LIN {X 0,Y 641.804,Z 360.991,A -85,B 0,C 180,E1 23081.821,E2 23081.821} C_VEL
LIN {X 0,Y 635.223,Z 347.429,A -85,B 0,C 180,E1 23079.954,E2 23079.954} C_VEL
LIN {X 0,Y 631.078,Z 339.172,A -85,B 0,C 180,E1 23078.744,E2 23078.744} C_VEL
LIN {X 0,Y 626.769,Z 330.556,A -85,B 0,C 180,E1 23077.432,E2 23077.432} C_VEL
LIN {X 0,Y 625.015,Z 327.05,A -85,B 0,C 180,E1 23076.864,E2 23076.864} C_VEL
LIN {X 0,Y 624.908,Z 326.441,A -85,B 0,C 180,E1 23076.643,E2 23076.643} C_VEL
LIN {X 0,Y 624.949,Z 326.345,A -85,B 0,C 180,E1 23073.503,E2 23073.503} C_VEL
LIN {X 0,Y 624.913,Z 326.377,A -85,B 0,C 180,E1 23070.412,E2 23070.412} C_VEL
LIN {X 0,Y 624.947,Z 326.372,A -85,B 0,C 180,E1 23067.232,E2 23067.232} C_VEL
LIN {X 0,Y 624.931,Z 326.347,A -85,B 0,C 180,E1 23064.079,E2 23064.079} C_VEL
LIN {X 0,Y 624.933,Z 326.384,A -85,B 0,C 180,E1 23060.806,E2 23060.806} C_VEL
LIN {X 0,Y 624.947,Z 326.347,A -85,B 0,C 180,E1 23057.698,E2 23057.698} C_VEL
LIN {X 0,Y 624.931,Z 326.381,A -85,B 0,C 180,E1 23054.537,E2 23054.537} C_VEL
LIN {X 0,Y 624.939,Z 326.352,A -85,B 0,C 180,E1 23051.443,E2 23051.443} C_VEL
LIN {X 0,Y 624.935,Z 326.375,A -85,B 0,C 180,E1 23048.372,E2 23048.372} C_VEL
LIN {X 0,Y 624.93,Z 326.352,A -85,B 0,C 180,E1 23045.325,E2 23045.325} C_VEL
LIN {X 0,Y 624.94,Z 326.376,A -85,B 0,C 180,E1 23042.201,E2 23042.201} C_VEL
LIN {X 0,Y 624.923,Z 326.355,A -85,B 0,C 180,E1 23039.083,E2 23039.083} C_VEL
LIN {X 0,Y 624.944,Z 326.376,A -85,B 0,C 180,E1 23035.963,E2 23035.963} C_VEL
LIN {X 0,Y 624.915,Z 326.354,A -85,B 0,C 180,E1 23032.923,E2 23032.923} C_VEL
LIN {X 0,Y 624.949,Z 326.375,A -85,B 0,C 180,E1 23029.863,E2 23029.863} C_VEL
LIN {X 0,Y 624.908,Z 326.359,A -85,B 0,C 180,E1 23026.773,E2 23026.773} C_VEL
LIN {X 0,Y 624.953,Z 326.368,A -85,B 0,C 180,E1 23023.73,E2 23023.73} C_VEL
LIN {X 0,Y 624.903,Z 326.37,A -85,B 0,C 180,E1 23020.657,E2 23020.657} C_VEL
LIN {X 0,Y 624.955,Z 326.352,A -85,B 0,C 180,E1 23017.618,E2 23017.618} C_VEL
LIN {X 0,Y 624.896,Z 326.392,A -85,B 0,C 180,E1 23014.607,E2 23014.607} C_VEL
LIN {X 0,Y 624.957,Z 326.344,A -85,B 0,C 180,E1 23011.629,E2 23011.629} C_VEL
LIN {X 0,Y 624.888,Z 326.373,A -85,B 0,C 180,E1 23008.665,E2 23008.665} C_VEL
LIN {X 0,Y 624.913,Z 326.378,A -85,B 0,C 180,E1 23005.813,E2 23005.813} C_VEL
LIN {X 0,Y 624.927,Z 326.63,A -85,B 0,C 180,E1 23004.753,E2 23004.753} C_VEL
LIN {X 0,Y 626.262,Z 329.964,A -85,B 0,C 180,E1 23004.242,E2 23004.242} C_VEL
LIN {X 0,Y 627.651,Z 332.24,A -85,B 0,C 180,E1 23003.869,E2 23003.869} C_VEL
LIN {X 0,Y 630.344,Z 337.573,A -85,B 0,C 180,E1 23003.079,E2 23003.079} C_VEL
LIN {X 0,Y 636.416,Z 349.11,A -85,B 0,C 180,E1 23001.41,E2 23001.41} C_VEL
LIN {X 0,Y 638.709,Z 353.459,A -85,B 0,C 180,E1 23000.855,E2 23000.855} C_VEL
LIN {X 0,Y 656.316,Z 378.29,A -85,B 0,C 180,E1 22998.74,E2 22998.74} C_VEL
LIN {X 0,Y 661.405,Z 385.767,A -85,B 0,C 180,E1 22998.161,E2 22998.161} C_VEL
LIN {X 0,Y 657.846,Z 584.34,A -85,B 0,C 180,E1 22995.477,E2 22995.477} C_VEL
LIN {X 0,Y 653.631,Z 808.573,A -85,B 0,C 180,E1 22992.489,E2 22992.489} C_VEL
LIN {X 0,Y 652.607,Z 840.702,A -85,B 0,C 180,E1 22992.004,E2 22992.004} C_VEL
LIN {X 0,Y 651.456,Z 864.088,A -85,B 0,C 180,E1 22991.512,E2 22991.512} C_VEL
LIN {X 0,Y 650.123,Z 886.354,A -85,B 0,C 180,E1 22990.922,E2 22990.922} C_VEL
LIN {X 0,Y 648.327,Z 912.621,A -85,B 0,C 180,E1 22990.066,E2 22990.066} C_VEL
LIN {X 0,Y 646.181,Z 938.349,A -85,B 0,C 180,E1 22989.032,E2 22989.032} C_VEL
LIN {X 0,Y 644.374,Z 958.689,A -85,B 0,C 180,E1 22988.083,E2 22988.083} C_VEL
LIN {X 0,Y 642.408,Z 979.352,A -85,B 0,C 180,E1 22986.988,E2 22986.988} C_VEL
LIN {X 0,Y 639.991,Z 1003.732,A -85,B 0,C 180,E1 22985.512,E2 22985.512} C_VEL
LIN {X 0,Y 637.696,Z 1025.632,A -85,B 0,C 180,E1 22983.979,E2 22983.979} C_VEL
LIN {X 0,Y 635.819,Z 1043.504,A -85,B 0,C 180,E1 22982.583,E2 22982.583} C_VEL
LIN {X 0,Y 633.971,Z 1061.27,A -85,B 0,C 180,E1 22981.046,E2 22981.046} C_VEL
LIN {X 0,Y 631.756,Z 1082.664,A -85,B 0,C 180,E1 22978.967,E2 22978.967} C_VEL
LIN {X 0,Y 630.187,Z 1098.843,A -85,B 0,C 180,E1 22977.19,E2 22977.19} C_VEL
LIN {X 0,Y 628.766,Z 1114.163,A -85,B 0,C 180,E1 22975.326,E2 22975.326} C_VEL
LIN {X 0,Y 627.338,Z 1131.25,A -85,B 0,C 180,E1 22972.985,E2 22972.985} C_VEL
LIN {X 0,Y 626.314,Z 1144.859,A -85,B 0,C 180,E1 22970.855,E2 22970.855} C_VEL
LIN {X 0,Y 625.553,Z 1156.307,A -85,B 0,C 180,E1 22968.837,E2 22968.837} C_VEL
LIN {X 0,Y 624.897,Z 1168.201,A -85,B 0,C 180,E1 22966.452,E2 22966.452} C_VEL
LIN {X 0,Y 624.452,Z 1178.088,A -85,B 0,C 180,E1 22964.086,E2 22964.086} C_VEL
LIN {X 0,Y 624.187,Z 1185.798,A -85,B 0,C 180,E1 22961.926,E2 22961.926} C_VEL
LIN {X 0,Y 624.035,Z 1192.621,A -85,B 0,C 180,E1 22959.592,E2 22959.592} C_VEL
LIN {X 0,Y 623.952,Z 1198.251,A -85,B 0,C 180,E1 22957.088,E2 22957.088} C_VEL
LIN {X 0,Y 623.914,Z 1202.013,A -85,B 0,C 180,E1 22954.688,E2 22954.688} C_VEL
LIN {X 0,Y 623.909,Z 1204.208,A -85,B 0,C 180,E1 22952.388,E2 22952.388} C_VEL
LIN {X 0,Y 623.902,Z 1204.961,A -85,B 0,C 180,E1 22949.816,E2 22949.816} C_VEL
LIN {X 0,Y 623.908,Z 1204.072,A -85,B 0,C 180,E1 22947.428,E2 22947.428} C_VEL
LIN {X 0,Y 623.916,Z 1201.898,A -85,B 0,C 180,E1 22945.22,E2 22945.22} C_VEL
LIN {X 0,Y 623.957,Z 1198.078,A -85,B 0,C 180,E1 22942.819,E2 22942.819} C_VEL
LIN {X 0,Y 624.037,Z 1192.376,A -85,B 0,C 180,E1 22940.314,E2 22940.314} C_VEL
LIN {X 0,Y 624.193,Z 1185.493,A -85,B 0,C 180,E1 22937.98,E2 22937.98} C_VEL
LIN {X 0,Y 624.484,Z 1177.37,A -85,B 0,C 180,E1 22935.725,E2 22935.725} C_VEL
LIN {X 0,Y 624.975,Z 1166.372,A -85,B 0,C 180,E1 22933.167,E2 22933.167} C_VEL
LIN {X 0,Y 625.583,Z 1155.793,A -85,B 0,C 180,E1 22931.067,E2 22931.067} C_VEL
LIN {X 0,Y 626.354,Z 1144.276,A -85,B 0,C 180,E1 22929.048,E2 22929.048} C_VEL
LIN {X 0,Y 627.501,Z 1129.294,A -85,B 0,C 180,E1 22926.723,E2 22926.723} C_VEL
LIN {X 0,Y 628.841,Z 1113.387,A -85,B 0,C 180,E1 22924.576,E2 22924.576} C_VEL
LIN {X 0,Y 630.262,Z 1097.992,A -85,B 0,C 180,E1 22922.711,E2 22922.711} C_VEL
LIN {X 0,Y 632.179,Z 1078.816,A -85,B 0,C 180,E1 22920.633,E2 22920.633} C_VEL
LIN {X 0,Y 634.138,Z 1059.603,A -85,B 0,C 180,E1 22918.804,E2 22918.804} C_VEL
LIN {X 0,Y 635.95,Z 1042.219,A -85,B 0,C 180,E1 22917.311,E2 22917.311} C_VEL
LIN {X 0,Y 637.972,Z 1022.949,A -85,B 0,C 180,E1 22915.82,E2 22915.82} C_VEL
LIN {X 0,Y 640.482,Z 998.662,A -85,B 0,C 180,E1 22914.167,E2 22914.167} C_VEL
LIN {X 0,Y 642.581,Z 977.633,A -85,B 0,C 180,E1 22912.917,E2 22912.917} C_VEL
LIN {X 0,Y 644.476,Z 957.681,A -85,B 0,C 180,E1 22911.867,E2 22911.867} C_VEL
LIN {X 0,Y 646.516,Z 934.93,A -85,B 0,C 180,E1 22910.819,E2 22910.819} C_VEL
LIN {X 0,Y 648.637,Z 907.797,A -85,B 0,C 180,E1 22909.767,E2 22909.767} C_VEL
LIN {X 0,Y 650.225,Z 884.749,A -85,B 0,C 180,E1 22909.032,E2 22909.032} C_VEL
LIN {X 0,Y 651.542,Z 862.576,A -85,B 0,C 180,E1 22908.452,E2 22908.452} C_VEL
LIN {X 0,Y 652.811,Z 836.723,A -85,B 0,C 180,E1 22907.922,E2 22907.922} C_VEL
LIN {X 0,Y 653.818,Z 798.385,A -85,B 0,C 180,E1 22907.377,E2 22907.377} C_VEL
LIN {X 0,Y 658.111,Z 571.161,A -85,B 0,C 180,E1 22904.345,E2 22904.345} C_VEL
LIN {X 0,Y 661.359,Z 385.453,A -85,B 0,C 180,E1 22901.83,E2 22901.83} C_VEL
LIN {X 0,Y 644.698,Z 361.888,A -85,B 0,C 180,E1 22899.89,E2 22899.89} C_VEL
LIN {X 0,Y 638.077,Z 352.586,A -85,B 0,C 180,E1 22899.047,E2 22899.047} C_VEL
LIN {X 0,Y 633.374,Z 343.405,A -85,B 0,C 180,E1 22897.773,E2 22897.773} C_VEL
LIN {X 0,Y 628.853,Z 334.634,A -85,B 0,C 180,E1 22896.489,E2 22896.489} C_VEL
LIN {X 0,Y 626.609,Z 330.419,A -85,B 0,C 180,E1 22895.844,E2 22895.844} C_VEL
LIN {X 0,Y 624.978,Z 326.955,A -85,B 0,C 180,E1 22895.31,E2 22895.31} C_VEL
LIN {X 0,Y 624.918,Z 326.379,A -85,B 0,C 180,E1 22894.947,E2 22894.947} C_VEL
LIN {X 0,Y 624.888,Z 326.361,A -85,B 0,C 180,E1 22891.826,E2 22891.826} C_VEL
LIN {X 0,Y 624.899,Z 326.361,A -85,B 0,C 180,E1 22889.106,E2 22889.106} C_VEL
LIN {X 0,Y 624.906,Z 326.39,A -85,B 0,C 180,E1 22885.799,E2 22885.799} C_VEL
LIN {X 0,Y 624.915,Z 326.349,A -85,B 0,C 180,E1 22882.881,E2 22882.881} C_VEL
LIN {X 0,Y 624.911,Z 326.38,A -85,B 0,C 180,E1 22879.634,E2 22879.634} C_VEL
LIN {X 0,Y 624.94,Z 326.36,A -85,B 0,C 180,E1 22876.589,E2 22876.589} C_VEL
LIN {X 0,Y 624.912,Z 326.364,A -85,B 0,C 180,E1 22873.415,E2 22873.415} C_VEL
LIN {X 0,Y 624.949,Z 326.368,A -85,B 0,C 180,E1 22870.323,E2 22870.323} C_VEL
LIN {X 0,Y 624.914,Z 326.357,A -85,B 0,C 180,E1 22867.169,E2 22867.169} C_VEL
LIN {X 0,Y 624.947,Z 326.372,A -85,B 0,C 180,E1 22864.129,E2 22864.129} C_VEL
LIN {X 0,Y 624.919,Z 326.359,A -85,B 0,C 180,E1 22861.008,E2 22861.008} C_VEL
LIN {X 0,Y 624.941,Z 326.368,A -85,B 0,C 180,E1 22857.983,E2 22857.983} C_VEL
LIN {X 0,Y 624.927,Z 326.359,A -85,B 0,C 180,E1 22854.859,E2 22854.859} C_VEL
LIN {X 0,Y 624.935,Z 326.365,A -85,B 0,C 180,E1 22851.813,E2 22851.813} C_VEL
LIN {X 0,Y 624.934,Z 326.359,A -85,B 0,C 180,E1 22848.744,E2 22848.744} C_VEL
LIN {X 0,Y 624.93,Z 326.372,A -85,B 0,C 180,E1 22845.641,E2 22845.641} C_VEL
LIN {X 0,Y 624.939,Z 326.355,A -85,B 0,C 180,E1 22842.591,E2 22842.591} C_VEL
LIN {X 0,Y 624.926,Z 326.384,A -85,B 0,C 180,E1 22839.488,E2 22839.488} C_VEL
LIN {X 0,Y 624.944,Z 326.347,A -85,B 0,C 180,E1 22836.422,E2 22836.422} C_VEL
LIN {X 0,Y 624.92,Z 326.387,A -85,B 0,C 180,E1 22833.384,E2 22833.384} C_VEL
LIN {X 0,Y 624.947,Z 326.35,A -85,B 0,C 180,E1 22830.316,E2 22830.316} C_VEL
LIN {X 0,Y 624.908,Z 326.356,A -85,B 0,C 180,E1 22827.312,E2 22827.312} C_VEL
LIN {X 0,Y 624.954,Z 326.378,A -85,B 0,C 180,E1 22824.21,E2 22824.21} C_VEL
LIN {X 0,Y 624.946,Z 326.651,A -85,B 0,C 180,E1 22823.105,E2 22823.105} C_VEL
LIN {X 0,Y 626.468,Z 330.148,A -85,B 0,C 180,E1 22822.547,E2 22822.547} C_VEL
LIN {X 0,Y 627.637,Z 332.307,A -85,B 0,C 180,E1 22822.201,E2 22822.201} C_VEL
LIN {X 0,Y 634.063,Z 344.875,A -85,B 0,C 180,E1 22820.307,E2 22820.307} C_VEL
LIN {X 0,Y 641.872,Z 361.171,A -85,B 0,C 180,E1 22818.065,E2 22818.065} C_VEL
LIN {X 0,Y 649.819,Z 378.958,A -85,B 0,C 180,E1 22815.837,E2 22815.837} C_VEL
LIN {X 0,Y 648.792,Z 394.463,A -85,B 0,C 180,E1 22814.752,E2 22814.752} C_VEL
LIN {X 0,Y 650.304,Z 401.327,A -85,B 0,C 180,E1 22814.502,E2 22814.502} C_VEL
LIN {X 0,Y 651.352,Z 408.644,A -85,B 0,C 180,E1 22814.292,E2 22814.292} C_VEL
LIN {X 0,Y 651.333,Z 419.658,A -85,B 0,C 180,E1 22814.125,E2 22814.125} C_VEL
LIN {X 0,Y 650.372,Z 436.541,A -85,B 0,C 180,E1 22813.955,E2 22813.955} C_VEL
LIN {X 0,Y 645.669,Z 670.245,A -85,B 0,C 180,E1 22810.849,E2 22810.849} C_VEL
LIN {X 0,Y 642.293,Z 830.084,A -85,B 0,C 180,E1 22808.725,E2 22808.725} C_VEL
LIN {X 0,Y 641.163,Z 856.269,A -85,B 0,C 180,E1 22808.241,E2 22808.241} C_VEL
LIN {X 0,Y 639.753,Z 879.486,A -85,B 0,C 180,E1 22807.648,E2 22807.648} C_VEL
LIN {X 0,Y 638.346,Z 899.141,A -85,B 0,C 180,E1 22807.032,E2 22807.032} C_VEL
LIN {X 0,Y 636.661,Z 920.113,A -85,B 0,C 180,E1 22806.249,E2 22806.249} C_VEL
LIN {X 0,Y 634.578,Z 944.969,A -85,B 0,C 180,E1 22805.158,E2 22805.158} C_VEL
LIN {X 0,Y 632.686,Z 965.707,A -85,B 0,C 180,E1 22804.093,E2 22804.093} C_VEL
LIN {X 0,Y 630.876,Z 984.683,A -85,B 0,C 180,E1 22802.985,E2 22802.985} C_VEL
LIN {X 0,Y 628.583,Z 1007.653,A -85,B 0,C 180,E1 22801.45,E2 22801.45} C_VEL
LIN {X 0,Y 626.685,Z 1026.358,A -85,B 0,C 180,E1 22800.013,E2 22800.013} C_VEL
LIN {X 0,Y 624.97,Z 1043.343,A -85,B 0,C 180,E1 22798.556,E2 22798.556} C_VEL
LIN {X 0,Y 622.908,Z 1063.939,A -85,B 0,C 180,E1 22796.554,E2 22796.554} C_VEL
LIN {X 0,Y 621.441,Z 1079.527,A -85,B 0,C 180,E1 22794.831,E2 22794.831} C_VEL
LIN {X 0,Y 619.965,Z 1096.148,A -85,B 0,C 180,E1 22792.773,E2 22792.773} C_VEL
LIN {X 0,Y 618.758,Z 1110.872,A -85,B 0,C 180,E1 22790.667,E2 22790.667} C_VEL
LIN {X 0,Y 617.877,Z 1123.126,A -85,B 0,C 180,E1 22788.688,E2 22788.688} C_VEL
LIN {X 0,Y 617.093,Z 1136.012,A -85,B 0,C 180,E1 22786.279,E2 22786.279} C_VEL
LIN {X 0,Y 616.619,Z 1145.191,A -85,B 0,C 180,E1 22784.269,E2 22784.269} C_VEL
LIN {X 0,Y 616.299,Z 1153.404,A -85,B 0,C 180,E1 22782.176,E2 22782.176} C_VEL
LIN {X 0,Y 616.061,Z 1161.254,A -85,B 0,C 180,E1 22779.718,E2 22779.718} C_VEL
LIN {X 0,Y 615.977,Z 1166.228,A -85,B 0,C 180,E1 22777.743,E2 22777.743} C_VEL
LIN {X 0,Y 615.913,Z 1170.071,A -85,B 0,C 180,E1 22775.777,E2 22775.777} C_VEL
LIN {X 0,Y 615.902,Z 1173.027,A -85,B 0,C 180,E1 22773.63,E2 22773.63} C_VEL
LIN {X 0,Y 615.911,Z 1174.701,A -85,B 0,C 180,E1 22771.209,E2 22771.209} C_VEL
LIN {X 0,Y 615.901,Z 1174.814,A -85,B 0,C 180,E1 22769.163,E2 22769.163} C_VEL
LIN {X 0,Y 615.906,Z 1173.836,A -85,B 0,C 180,E1 22767.209,E2 22767.209} C_VEL
LIN {X 0,Y 615.921,Z 1171.322,A -85,B 0,C 180,E1 22764.878,E2 22764.878} C_VEL
LIN {X 0,Y 615.961,Z 1167.047,A -85,B 0,C 180,E1 22762.539,E2 22762.539} C_VEL
LIN {X 0,Y 616.053,Z 1162.263,A -85,B 0,C 180,E1 22760.565,E2 22760.565} C_VEL
LIN {X 0,Y 616.21,Z 1156.003,A -85,B 0,C 180,E1 22758.488,E2 22758.488} C_VEL
LIN {X 0,Y 616.555,Z 1146.792,A -85,B 0,C 180,E1 22756.017,E2 22756.017} C_VEL
LIN {X 0,Y 616.992,Z 1137.822,A -85,B 0,C 180,E1 22754.009,E2 22754.009} C_VEL
LIN {X 0,Y 617.591,Z 1127.457,A -85,B 0,C 180,E1 22751.988,E2 22751.988} C_VEL
LIN {X 0,Y 618.549,Z 1113.531,A -85,B 0,C 180,E1 22749.649,E2 22749.649} C_VEL
LIN {X 0,Y 619.608,Z 1100.314,A -85,B 0,C 180,E1 22747.715,E2 22747.715} C_VEL
LIN {X 0,Y 620.996,Z 1084.506,A -85,B 0,C 180,E1 22745.658,E2 22745.658} C_VEL
LIN {X 0,Y 622.612,Z 1067.07,A -85,B 0,C 180,E1 22743.69,E2 22743.69} C_VEL
LIN {X 0,Y 624.168,Z 1051.184,A -85,B 0,C 180,E1 22742.083,E2 22742.083} C_VEL
LIN {X 0,Y 626.351,Z 1029.845,A -85,B 0,C 180,E1 22740.181,E2 22740.181} C_VEL
LIN {X 0,Y 628.199,Z 1011.463,A -85,B 0,C 180,E1 22738.743,E2 22738.743} C_VEL
LIN {X 0,Y 630.281,Z 990.792,A -85,B 0,C 180,E1 22737.305,E2 22737.305} C_VEL
LIN {X 0,Y 632.479,Z 967.857,A -85,B 0,C 180,E1 22735.935,E2 22735.935} C_VEL
LIN {X 0,Y 634.238,Z 948.527,A -85,B 0,C 180,E1 22734.926,E2 22734.926} C_VEL
LIN {X 0,Y 636.336,Z 924.605,A -85,B 0,C 180,E1 22733.842,E2 22733.842} C_VEL
LIN {X 0,Y 638.238,Z 900.726,A -85,B 0,C 180,E1 22732.933,E2 22732.933} C_VEL
LIN {X 0,Y 639.672,Z 880.707,A -85,B 0,C 180,E1 22732.298,E2 22732.298} C_VEL
LIN {X 0,Y 640.897,Z 860.874,A -85,B 0,C 180,E1 22731.78,E2 22731.78} C_VEL
LIN {X 0,Y 642.142,Z 836.025,A -85,B 0,C 180,E1 22731.276,E2 22731.276} C_VEL
LIN {X 0,Y 643.231,Z 791.041,A -85,B 0,C 180,E1 22730.653,E2 22730.653} C_VEL
LIN {X 0,Y 647.657,Z 571.402,A -85,B 0,C 180,E1 22727.75,E2 22727.75} C_VEL
LIN {X 0,Y 650.402,Z 429.922,A -85,B 0,C 180,E1 22725.856,E2 22725.856} C_VEL
LIN {X 0,Y 642.675,Z 393.196,A -85,B 0,C 180,E1 22724.529,E2 22724.529} C_VEL
LIN {X 0,Y 643.362,Z 382.663,A -85,B 0,C 180,E1 22723.757,E2 22723.757} C_VEL
LIN {X 0,Y 635.717,Z 365.668,A -85,B 0,C 180,E1 22721.586,E2 22721.586} C_VEL
LIN {X 0,Y 629.219,Z 352.169,A -85,B 0,C 180,E1 22719.704,E2 22719.704} C_VEL
LIN {X 0,Y 625.087,Z 343.962,A -85,B 0,C 180,E1 22718.481,E2 22718.481} C_VEL
LIN {X 0,Y 621.118,Z 336.002,A -85,B 0,C 180,E1 22717.25,E2 22717.25} C_VEL
LIN {X 0,Y 618.676,Z 331.391,A -85,B 0,C 180,E1 22716.495,E2 22716.495} C_VEL
LIN {X 0,Y 617.071,Z 327.744,A -85,B 0,C 180,E1 22715.904,E2 22715.904} C_VEL
LIN {X 0,Y 616.966,Z 327.366,A -85,B 0,C 180,E1 22714.911,E2 22714.911} C_VEL
LIN {X 0,Y 617.011,Z 327.356,A -85,B 0,C 180,E1 22711.881,E2 22711.881} C_VEL
LIN {X 0,Y 616.968,Z 327.335,A -85,B 0,C 180,E1 22708.747,E2 22708.747} C_VEL
LIN {X 0,Y 617.012,Z 327.364,A -85,B 0,C 180,E1 22705.638,E2 22705.638} C_VEL
LIN {X 0,Y 616.978,Z 327.356,A -85,B 0,C 180,E1 22702.487,E2 22702.487} C_VEL
LIN {X 0,Y 617.004,Z 327.34,A -85,B 0,C 180,E1 22699.403,E2 22699.403} C_VEL
LIN {X 0,Y 616.988,Z 327.368,A -85,B 0,C 180,E1 22696.282,E2 22696.282} C_VEL
LIN {X 0,Y 616.999,Z 327.33,A -85,B 0,C 180,E1 22693.209,E2 22693.209} C_VEL
LIN {X 0,Y 617,Z 327.369,A -85,B 0,C 180,E1 22689.986,E2 22689.986} C_VEL
LIN {X 0,Y 617.006,Z 327.324,A -85,B 0,C 180,E1 22686.794,E2 22686.794} C_VEL
LIN {X 0,Y 617.005,Z 327.375,A -85,B 0,C 180,E1 22683.531,E2 22683.531} C_VEL
LIN {X 0,Y 617.003,Z 327.325,A -85,B 0,C 180,E1 22680.279,E2 22680.279} C_VEL
LIN {X 0,Y 616.987,Z 327.376,A -85,B 0,C 180,E1 22677.12,E2 22677.12} C_VEL
LIN {X 0,Y 617.003,Z 327.327,A -85,B 0,C 180,E1 22673.953,E2 22673.953} C_VEL
LIN {X 0,Y 616.977,Z 327.374,A -85,B 0,C 180,E1 22670.861,E2 22670.861} C_VEL
LIN {X 0,Y 617.008,Z 327.327,A -85,B 0,C 180,E1 22667.734,E2 22667.734} C_VEL
LIN {X 0,Y 616.972,Z 327.375,A -85,B 0,C 180,E1 22664.636,E2 22664.636} C_VEL
LIN {X 0,Y 617.006,Z 327.332,A -85,B 0,C 180,E1 22661.443,E2 22661.443} C_VEL
LIN {X 0,Y 616.967,Z 327.369,A -85,B 0,C 180,E1 22658.414,E2 22658.414} C_VEL
LIN {X 0,Y 616.99,Z 327.358,A -85,B 0,C 180,E1 22655.182,E2 22655.182} C_VEL
LIN {X 0,Y 616.956,Z 327.341,A -85,B 0,C 180,E1 22652.236,E2 22652.236} C_VEL
LIN {X 0,Y 616.977,Z 327.368,A -85,B 0,C 180,E1 22649.014,E2 22649.014} C_VEL
LIN {X 0,Y 616.948,Z 327.358,A -85,B 0,C 180,E1 22646.115,E2 22646.115} C_VEL
LIN {X 0,Y 617.067,Z 327.839,A -85,B 0,C 180,E1 22645.631,E2 22645.631} C_VEL
LIN {X 0,Y 618.571,Z 331.239,A -85,B 0,C 180,E1 22645.094,E2 22645.094} C_VEL
LIN {X 0,Y 619.563,Z 332.834,A -85,B 0,C 180,E1 22644.82,E2 22644.82} C_VEL
LIN {X 0,Y 621.413,Z 336.398,A -85,B 0,C 180,E1 22644.261,E2 22644.261} C_VEL
LIN {X 0,Y 624.861,Z 343.132,A -85,B 0,C 180,E1 22643.24,E2 22643.24} C_VEL
LIN {X 0,Y 630.41,Z 353.7,A -85,B 0,C 180,E1 22641.719,E2 22641.719} C_VEL
LIN {X 0,Y 642.453,Z 370.467,A -85,B 0,C 180,E1 22640.189,E2 22640.189} C_VEL
LIN {X 0,Y 655.762,Z 389.515,A -85,B 0,C 180,E1 22638.614,E2 22638.614} C_VEL
LIN {X 0,Y 651.89,Z 597.338,A -85,B 0,C 180,E1 22635.798,E2 22635.798} C_VEL
LIN {X 0,Y 647.542,Z 817.265,A -85,B 0,C 180,E1 22632.851,E2 22632.851} C_VEL
LIN {X 0,Y 646.533,Z 843.059,A -85,B 0,C 180,E1 22632.436,E2 22632.436} C_VEL
LIN {X 0,Y 645.363,Z 865.27,A -85,B 0,C 180,E1 22631.958,E2 22631.958} C_VEL
LIN {X 0,Y 643.909,Z 888.073,A -85,B 0,C 180,E1 22631.344,E2 22631.344} C_VEL
LIN {X 0,Y 641.792,Z 916.153,A -85,B 0,C 180,E1 22630.399,E2 22630.399} C_VEL
LIN {X 0,Y 639.767,Z 939.13,A -85,B 0,C 180,E1 22629.459,E2 22629.459} C_VEL
LIN {X 0,Y 637.82,Z 959.692,A -85,B 0,C 180,E1 22628.488,E2 22628.488} C_VEL
LIN {X 0,Y 635.634,Z 981.239,A -85,B 0,C 180,E1 22627.33,E2 22627.33} C_VEL
LIN {X 0,Y 632.927,Z 1006.383,A -85,B 0,C 180,E1 22625.768,E2 22625.768} C_VEL
LIN {X 0,Y 630.713,Z 1026.231,A -85,B 0,C 180,E1 22624.358,E2 22624.358} C_VEL
LIN {X 0,Y 628.715,Z 1044.05,A -85,B 0,C 180,E1 22622.949,E2 22622.949} C_VEL
LIN {X 0,Y 626.621,Z 1062.931,A -85,B 0,C 180,E1 22621.291,E2 22621.291} C_VEL
LIN {X 0,Y 624.267,Z 1083.985,A -85,B 0,C 180,E1 22619.199,E2 22619.199} C_VEL
LIN {X 0,Y 622.628,Z 1099.686,A -85,B 0,C 180,E1 22617.444,E2 22617.444} C_VEL
LIN {X 0,Y 621.011,Z 1116.093,A -85,B 0,C 180,E1 22615.409,E2 22615.409} C_VEL
LIN {X 0,Y 619.468,Z 1133.186,A -85,B 0,C 180,E1 22612.992,E2 22612.992} C_VEL
LIN {X 0,Y 618.444,Z 1146.007,A -85,B 0,C 180,E1 22610.935,E2 22610.935} C_VEL
LIN {X 0,Y 617.578,Z 1158.364,A -85,B 0,C 180,E1 22608.697,E2 22608.697} C_VEL
LIN {X 0,Y 616.881,Z 1170.26,A -85,B 0,C 180,E1 22606.188,E2 22606.188} C_VEL
LIN {X 0,Y 616.475,Z 1178.804,A -85,B 0,C 180,E1 22604.081,E2 22604.081} C_VEL
LIN {X 0,Y 616.204,Z 1186.098,A -85,B 0,C 180,E1 22601.987,E2 22601.987} C_VEL
LIN {X 0,Y 616.039,Z 1193.109,A -85,B 0,C 180,E1 22599.529,E2 22599.529} C_VEL
LIN {X 0,Y 615.947,Z 1198.595,A -85,B 0,C 180,E1 22596.993,E2 22596.993} C_VEL
LIN {X 0,Y 615.914,Z 1202.124,A -85,B 0,C 180,E1 22594.656,E2 22594.656} C_VEL
LIN {X 0,Y 615.911,Z 1204.27,A -85,B 0,C 180,E1 22592.326,E2 22592.326} C_VEL
LIN {X 0,Y 615.897,Z 1204.939,A -85,B 0,C 180,E1 22589.721,E2 22589.721} C_VEL
LIN {X 0,Y 615.909,Z 1204.069,A -85,B 0,C 180,E1 22587.394,E2 22587.394} C_VEL
LIN {X 0,Y 615.919,Z 1201.895,A -85,B 0,C 180,E1 22585.157,E2 22585.157} C_VEL
LIN {X 0,Y 615.961,Z 1197.988,A -85,B 0,C 180,E1 22582.676,E2 22582.676} C_VEL
LIN {X 0,Y 616.053,Z 1192.224,A -85,B 0,C 180,E1 22580.131,E2 22580.131} C_VEL
LIN {X 0,Y 616.221,Z 1185.489,A -85,B 0,C 180,E1 22577.823,E2 22577.823} C_VEL
LIN {X 0,Y 616.551,Z 1177.268,A -85,B 0,C 180,E1 22575.51,E2 22575.51} C_VEL
LIN {X 0,Y 617.08,Z 1166.361,A -85,B 0,C 180,E1 22572.943,E2 22572.943} C_VEL
LIN {X 0,Y 617.737,Z 1155.792,A -85,B 0,C 180,E1 22570.817,E2 22570.817} C_VEL
LIN {X 0,Y 618.571,Z 1144.279,A -85,B 0,C 180,E1 22568.772,E2 22568.772} C_VEL
LIN {X 0,Y 619.83,Z 1129.091,A -85,B 0,C 180,E1 22566.389,E2 22566.389} C_VEL
LIN {X 0,Y 621.28,Z 1113.387,A -85,B 0,C 180,E1 22564.244,E2 22564.244} C_VEL
LIN {X 0,Y 622.79,Z 1097.992,A -85,B 0,C 180,E1 22562.355,E2 22562.355} C_VEL
LIN {X 0,Y 624.875,Z 1078.873,A -85,B 0,C 180,E1 22560.262,E2 22560.262} C_VEL
LIN {X 0,Y 626.911,Z 1060.157,A -85,B 0,C 180,E1 22558.457,E2 22558.457} C_VEL
LIN {X 0,Y 628.846,Z 1042.825,A -85,B 0,C 180,E1 22556.949,E2 22556.949} C_VEL
LIN {X 0,Y 630.917,Z 1024.335,A -85,B 0,C 180,E1 22555.499,E2 22555.499} C_VEL
LIN {X 0,Y 633.603,Z 1000.27,A -85,B 0,C 180,E1 22553.828,E2 22553.828} C_VEL
LIN {X 0,Y 635.916,Z 978.529,A -85,B 0,C 180,E1 22552.519,E2 22552.519} C_VEL
LIN {X 0,Y 637.938,Z 958.565,A -85,B 0,C 180,E1 22551.456,E2 22551.456} C_VEL
LIN {X 0,Y 639.965,Z 937.188,A -85,B 0,C 180,E1 22550.455,E2 22550.455} C_VEL
LIN {X 0,Y 642.289,Z 910.008,A -85,B 0,C 180,E1 22549.375,E2 22549.375} C_VEL
LIN {X 0,Y 644.07,Z 885.61,A -85,B 0,C 180,E1 22548.584,E2 22548.584} C_VEL
LIN {X 0,Y 645.453,Z 863.751,A -85,B 0,C 180,E1 22548.005,E2 22548.005} C_VEL
LIN {X 0,Y 646.662,Z 840.442,A -85,B 0,C 180,E1 22547.514,E2 22547.514} C_VEL
LIN {X 0,Y 647.773,Z 806.479,A -85,B 0,C 180,E1 22547.004,E2 22547.004} C_VEL
LIN {X 0,Y 652.066,Z 587.341,A -85,B 0,C 180,E1 22544.07,E2 22544.07} C_VEL
LIN {X 0,Y 655.752,Z 389.473,A -85,B 0,C 180,E1 22541.385,E2 22541.385} C_VEL
LIN {X 0,Y 640.759,Z 368.06,A -85,B 0,C 180,E1 22539.603,E2 22539.603} C_VEL
LIN {X 0,Y 630.124,Z 353.272,A -85,B 0,C 180,E1 22538.233,E2 22538.233} C_VEL
LIN {X 0,Y 623.275,Z 340.031,A -85,B 0,C 180,E1 22536.297,E2 22536.297} C_VEL
LIN {X 0,Y 621.401,Z 336.386,A -85,B 0,C 180,E1 22535.74,E2 22535.74} C_VEL
LIN {X 0,Y 618.914,Z 331.695,A -85,B 0,C 180,E1 22534.996,E2 22534.996} C_VEL
LIN {X 0,Y 617.1,Z 327.993,A -85,B 0,C 180,E1 22534.396,E2 22534.396} C_VEL
LIN {X 0,Y 616.968,Z 327.401,A -85,B 0,C 180,E1 22534.091,E2 22534.091} C_VEL
LIN {X 0,Y 616.952,Z 327.362,A -85,B 0,C 180,E1 22531.24,E2 22531.24} C_VEL
LIN {X 0,Y 616.977,Z 327.336,A -85,B 0,C 180,E1 22528.033,E2 22528.033} C_VEL
LIN {X 0,Y 616.962,Z 327.371,A -85,B 0,C 180,E1 22525.126,E2 22525.126} C_VEL
LIN {X 0,Y 616.986,Z 327.355,A -85,B 0,C 180,E1 22521.885,E2 22521.885} C_VEL
LIN {X 0,Y 616.974,Z 327.343,A -85,B 0,C 180,E1 22518.913,E2 22518.913} C_VEL
LIN {X 0,Y 616.983,Z 327.374,A -85,B 0,C 180,E1 22515.606,E2 22515.606} C_VEL
LIN {X 0,Y 616.999,Z 327.33,A -85,B 0,C 180,E1 22512.542,E2 22512.542} C_VEL
LIN {X 0,Y 616.979,Z 327.373,A -85,B 0,C 180,E1 22509.327,E2 22509.327} C_VEL
LIN {X 0,Y 617.007,Z 327.326,A -85,B 0,C 180,E1 22506.233,E2 22506.233} C_VEL
LIN {X 0,Y 616.983,Z 327.374,A -85,B 0,C 180,E1 22503.066,E2 22503.066} C_VEL
LIN {X 0,Y 617,Z 327.325,A -85,B 0,C 180,E1 22500,E2 22500} C_VEL
LIN {X 0,Y 616.989,Z 327.372,A -85,B 0,C 180,E1 22496.841,E2 22496.841} C_VEL
LIN {X 0,Y 616.995,Z 327.323,A -85,B 0,C 180,E1 22493.767,E2 22493.767} C_VEL
LIN {X 0,Y 616.997,Z 327.37,A -85,B 0,C 180,E1 22490.674,E2 22490.674} C_VEL
LIN {X 0,Y 616.991,Z 327.325,A -85,B 0,C 180,E1 22487.553,E2 22487.553} C_VEL
LIN {X 0,Y 617.005,Z 327.376,A -85,B 0,C 180,E1 22484.394,E2 22484.394} C_VEL
LIN {X 0,Y 616.997,Z 327.331,A -85,B 0,C 180,E1 22481.186,E2 22481.186} C_VEL
LIN {X 0,Y 617.002,Z 327.363,A -85,B 0,C 180,E1 22477.916,E2 22477.916} C_VEL
LIN {X 0,Y 617.011,Z 327.355,A -85,B 0,C 180,E1 22474.67,E2 22474.67} C_VEL
LIN {X 0,Y 616.977,Z 327.336,A -85,B 0,C 180,E1 22471.545,E2 22471.545} C_VEL
LIN {X 0,Y 617.015,Z 327.368,A -85,B 0,C 180,E1 22468.437,E2 22468.437} C_VEL
LIN {X 0,Y 616.97,Z 327.355,A -85,B 0,C 180,E1 22465.33,E2 22465.33} C_VEL
LIN {X 0,Y 617.053,Z 327.64,A -85,B 0,C 180,E1 22464.027,E2 22464.027} C_VEL
LIN {X 0,Y 618.438,Z 331.059,A -85,B 0,C 180,E1 22463.47,E2 22463.47} C_VEL
LIN {X 0,Y 619.646,Z 333.168,A -85,B 0,C 180,E1 22463.11,E2 22463.11} C_VEL
LIN {X 0,Y 622.372,Z 338.529,A -85,B 0,C 180,E1 22462.258,E2 22462.258} C_VEL
LIN {X 0,Y 628.667,Z 350.953,A -85,B 0,C 180,E1 22460.373,E2 22460.373} C_VEL
LIN {X 0,Y 636.126,Z 366.529,A -85,B 0,C 180,E1 22458.205,E2 22458.205} C_VEL
LIN {X 0,Y 643.455,Z 382.857,A -85,B 0,C 180,E1 22456.127,E2 22456.127} C_VEL
LIN {X 0,Y 642.764,Z 394.124,A -85,B 0,C 180,E1 22455.336,E2 22455.336} C_VEL
LIN {X 0,Y 650.497,Z 430.448,A -85,B 0,C 180,E1 22454.036,E2 22454.036} C_VEL
LIN {X 0,Y 650.372,Z 436.541,A -85,B 0,C 180,E1 22453.955,E2 22453.955} C_VEL
LIN {X 0,Y 649.526,Z 444.248,A -85,B 0,C 180,E1 22453.915,E2 22453.915} C_VEL
LIN {X 0,Y 644.786,Z 464.912,A -85,B 0,C 180,E1 22454.038,E2 22454.038} C_VEL
LIN {X 0,Y 644.124,Z 471.524,A -85,B 0,C 180,E1 22453.998,E2 22453.998} C_VEL
LIN {X 0,Y 639.301,Z 700.686,A -85,B 0,C 180,E1 22450.948,E2 22450.948} C_VEL
LIN {X 0,Y 636.406,Z 830.215,A -85,B 0,C 180,E1 22449.214,E2 22449.214} C_VEL
LIN {X 0,Y 635.215,Z 856.295,A -85,B 0,C 180,E1 22448.73,E2 22448.73} C_VEL
LIN {X 0,Y 633.705,Z 879.702,A -85,B 0,C 180,E1 22448.128,E2 22448.128} C_VEL
LIN {X 0,Y 632.16,Z 900.057,A -85,B 0,C 180,E1 22447.485,E2 22447.485} C_VEL
LIN {X 0,Y 630.237,Z 922.796,A -85,B 0,C 180,E1 22446.622,E2 22446.622} C_VEL
LIN {X 0,Y 627.92,Z 946.477,A -85,B 0,C 180,E1 22445.536,E2 22445.536} C_VEL
LIN {X 0,Y 625.61,Z 968.774,A -85,B 0,C 180,E1 22444.346,E2 22444.346} C_VEL
LIN {X 0,Y 623.155,Z 992.507,A -85,B 0,C 180,E1 22442.898,E2 22442.898} C_VEL
LIN {X 0,Y 621.103,Z 1011.666,A -85,B 0,C 180,E1 22441.547,E2 22441.547} C_VEL
LIN {X 0,Y 619.2,Z 1029.405,A -85,B 0,C 180,E1 22440.146,E2 22440.146} C_VEL
LIN {X 0,Y 616.892,Z 1050.579,A -85,B 0,C 180,E1 22438.248,E2 22438.248} C_VEL
LIN {X 0,Y 615.135,Z 1067.183,A -85,B 0,C 180,E1 22436.552,E2 22436.552} C_VEL
LIN {X 0,Y 613.415,Z 1084.647,A -85,B 0,C 180,E1 22434.554,E2 22434.554} C_VEL
LIN {X 0,Y 611.912,Z 1100.384,A -85,B 0,C 180,E1 22432.48,E2 22432.48} C_VEL
LIN {X 0,Y 610.775,Z 1113.675,A -85,B 0,C 180,E1 22430.508,E2 22430.508} C_VEL
LIN {X 0,Y 609.706,Z 1128.021,A -85,B 0,C 180,E1 22428.056,E2 22428.056} C_VEL
LIN {X 0,Y 609.062,Z 1138.312,A -85,B 0,C 180,E1 22426.01,E2 22426.01} C_VEL
LIN {X 0,Y 608.548,Z 1148.429,A -85,B 0,C 180,E1 22423.686,E2 22423.686} C_VEL
LIN {X 0,Y 608.21,Z 1156.63,A -85,B 0,C 180,E1 22421.378,E2 22421.378} C_VEL
LIN {X 0,Y 608.059,Z 1162.529,A -85,B 0,C 180,E1 22419.369,E2 22419.369} C_VEL
LIN {X 0,Y 607.967,Z 1167.471,A -85,B 0,C 180,E1 22417.275,E2 22417.275} C_VEL
LIN {X 0,Y 607.903,Z 1171.78,A -85,B 0,C 180,E1 22414.718,E2 22414.718} C_VEL
LIN {X 0,Y 607.905,Z 1173.904,A -85,B 0,C 180,E1 22412.64,E2 22412.64} C_VEL
LIN {X 0,Y 607.895,Z 1174.837,A -85,B 0,C 180,E1 22410.66,E2 22410.66} C_VEL
LIN {X 0,Y 607.908,Z 1174.656,A -85,B 0,C 180,E1 22408.492,E2 22408.492} C_VEL
LIN {X 0,Y 607.913,Z 1172.798,A -85,B 0,C 180,E1 22406.039,E2 22406.039} C_VEL
LIN {X 0,Y 607.923,Z 1170.062,A -85,B 0,C 180,E1 22404.053,E2 22404.053} C_VEL
LIN {X 0,Y 607.992,Z 1166.22,A -85,B 0,C 180,E1 22402.06,E2 22402.06} C_VEL
LIN {X 0,Y 608.09,Z 1160.732,A -85,B 0,C 180,E1 22399.867,E2 22399.867} C_VEL
LIN {X 0,Y 608.351,Z 1153.031,A -85,B 0,C 180,E1 22397.47,E2 22397.47} C_VEL
LIN {X 0,Y 608.692,Z 1145.166,A -85,B 0,C 180,E1 22395.444,E2 22395.444} C_VEL
LIN {X 0,Y 609.192,Z 1135.978,A -85,B 0,C 180,E1 22393.406,E2 22393.406} C_VEL
LIN {X 0,Y 610.05,Z 1123.078,A -85,B 0,C 180,E1 22390.964,E2 22390.964} C_VEL
LIN {X 0,Y 610.988,Z 1111.071,A -85,B 0,C 180,E1 22388.999,E2 22388.999} C_VEL
LIN {X 0,Y 612.241,Z 1096.784,A -85,B 0,C 180,E1 22386.924,E2 22386.924} C_VEL
LIN {X 0,Y 613.822,Z 1080.272,A -85,B 0,C 180,E1 22384.84,E2 22384.84} C_VEL
LIN {X 0,Y 615.346,Z 1065.126,A -85,B 0,C 180,E1 22383.137,E2 22383.137} C_VEL
LIN {X 0,Y 617.39,Z 1046.284,A -85,B 0,C 180,E1 22381.25,E2 22381.25} C_VEL
LIN {X 0,Y 619.404,Z 1027.396,A -85,B 0,C 180,E1 22379.598,E2 22379.598} C_VEL
LIN {X 0,Y 621.374,Z 1009.133,A -85,B 0,C 180,E1 22378.173,E2 22378.173} C_VEL
LIN {X 0,Y 623.937,Z 985.22,A -85,B 0,C 180,E1 22376.546,E2 22376.546} C_VEL
LIN {X 0,Y 626.108,Z 964.154,A -85,B 0,C 180,E1 22375.303,E2 22375.303} C_VEL
LIN {X 0,Y 628.756,Z 937.929,A -85,B 0,C 180,E1 22373.957,E2 22373.957} C_VEL
LIN {X 0,Y 630.754,Z 916.414,A -85,B 0,C 180,E1 22373.031,E2 22373.031} C_VEL
LIN {X 0,Y 632.614,Z 894.312,A -85,B 0,C 180,E1 22372.227,E2 22372.227} C_VEL
LIN {X 0,Y 634.503,Z 868.021,A -85,B 0,C 180,E1 22371.465,E2 22371.465} C_VEL
LIN {X 0,Y 635.689,Z 846.853,A -85,B 0,C 180,E1 22370.989,E2 22370.989} C_VEL
LIN {X 0,Y 636.604,Z 824.76,A -85,B 0,C 180,E1 22370.614,E2 22370.614} C_VEL
LIN {X 0,Y 641.081,Z 616.325,A -85,B 0,C 180,E1 22367.843,E2 22367.843} C_VEL
LIN {X 0,Y 644.882,Z 432.051,A -85,B 0,C 180,E1 22365.372,E2 22365.372} C_VEL
LIN {X 0,Y 636.68,Z 392.67,A -85,B 0,C 180,E1 22363.921,E2 22363.921} C_VEL
LIN {X 0,Y 637.086,Z 386.905,A -85,B 0,C 180,E1 22363.495,E2 22363.495} C_VEL
LIN {X 0,Y 629.442,Z 369.946,A -85,B 0,C 180,E1 22361.291,E2 22361.291} C_VEL
LIN {X 0,Y 622.336,Z 354.817,A -85,B 0,C 180,E1 22359.155,E2 22359.155} C_VEL
LIN {X 0,Y 615.488,Z 341.421,A -85,B 0,C 180,E1 22357.064,E2 22357.064} C_VEL
LIN {X 0,Y 613.062,Z 336.833,A -85,B 0,C 180,E1 22356.302,E2 22356.302} C_VEL
LIN {X 0,Y 611.068,Z 332.74,A -85,B 0,C 180,E1 22355.628,E2 22355.628} C_VEL
LIN {X 0,Y 609.215,Z 329.325,A -85,B 0,C 180,E1 22355.017,E2 22355.017} C_VEL
LIN {X 0,Y 609.038,Z 328.455,A -85,B 0,C 180,E1 22354.829,E2 22354.829} C_VEL
LIN {X 0,Y 609.076,Z 328.346,A -85,B 0,C 180,E1 22351.749,E2 22351.749} C_VEL
LIN {X 0,Y 609.029,Z 328.322,A -85,B 0,C 180,E1 22348.646,E2 22348.646} C_VEL
LIN {X 0,Y 609.074,Z 328.351,A -85,B 0,C 180,E1 22345.579,E2 22345.579} C_VEL
LIN {X 0,Y 609.042,Z 328.345,A -85,B 0,C 180,E1 22342.389,E2 22342.389} C_VEL
LIN {X 0,Y 609.067,Z 328.323,A -85,B 0,C 180,E1 22339.267,E2 22339.267} C_VEL
LIN {X 0,Y 609.056,Z 328.358,A -85,B 0,C 180,E1 22336.108,E2 22336.108} C_VEL
LIN {X 0,Y 609.067,Z 328.312,A -85,B 0,C 180,E1 22332.901,E2 22332.901} C_VEL
LIN {X 0,Y 609.07,Z 328.364,A -85,B 0,C 180,E1 22329.64,E2 22329.64} C_VEL
LIN {X 0,Y 609.058,Z 328.31,A -85,B 0,C 180,E1 22326.41,E2 22326.41} C_VEL
LIN {X 0,Y 609.056,Z 328.362,A -85,B 0,C 180,E1 22323.2,E2 22323.2} C_VEL
LIN {X 0,Y 609.059,Z 328.312,A -85,B 0,C 180,E1 22320,E2 22320} C_VEL
LIN {X 0,Y 609.049,Z 328.363,A -85,B 0,C 180,E1 22316.894,E2 22316.894} C_VEL
LIN {X 0,Y 609.07,Z 328.312,A -85,B 0,C 180,E1 22313.685,E2 22313.685} C_VEL
LIN {X 0,Y 609.049,Z 328.361,A -85,B 0,C 180,E1 22310.551,E2 22310.551} C_VEL
LIN {X 0,Y 609.044,Z 328.321,A -85,B 0,C 180,E1 22307.195,E2 22307.195} C_VEL
LIN {X 0,Y 609.069,Z 328.355,A -85,B 0,C 180,E1 22304.088,E2 22304.088} C_VEL
LIN {X 0,Y 609.029,Z 328.334,A -85,B 0,C 180,E1 22300.93,E2 22300.93} C_VEL
LIN {X 0,Y 609.068,Z 328.334,A -85,B 0,C 180,E1 22297.917,E2 22297.917} C_VEL
LIN {X 0,Y 609.021,Z 328.363,A -85,B 0,C 180,E1 22294.731,E2 22294.731} C_VEL
LIN {X 0,Y 609.079,Z 328.317,A -85,B 0,C 180,E1 22291.631,E2 22291.631} C_VEL
LIN {X 0,Y 609.009,Z 328.344,A -85,B 0,C 180,E1 22288.621,E2 22288.621} C_VEL
LIN {X 0,Y 609.041,Z 328.577,A -85,B 0,C 180,E1 22286.673,E2 22286.673} C_VEL
LIN {X 0,Y 610.591,Z 332.211,A -85,B 0,C 180,E1 22286.054,E2 22286.054} C_VEL
LIN {X 0,Y 611.88,Z 334.277,A -85,B 0,C 180,E1 22285.683,E2 22285.683} C_VEL
LIN {X 0,Y 614.567,Z 339.568,A -85,B 0,C 180,E1 22284.833,E2 22284.833} C_VEL
LIN {X 0,Y 619.005,Z 347.803,A -85,B 0,C 180,E1 22283.527,E2 22283.527} C_VEL
LIN {X 0,Y 622.524,Z 354.59,A -85,B 0,C 180,E1 22282.559,E2 22282.559} C_VEL
LIN {X 0,Y 635.441,Z 372.283,A -85,B 0,C 180,E1 22280.862,E2 22280.862} C_VEL
LIN {X 0,Y 650.151,Z 393.263,A -85,B 0,C 180,E1 22279.075,E2 22279.075} C_VEL
LIN {X 0,Y 646.025,Z 596.674,A -85,B 0,C 180,E1 22276.29,E2 22276.29} C_VEL
LIN {X 0,Y 642.646,Z 771.19,A -85,B 0,C 180,E1 22273.958,E2 22273.958} C_VEL
LIN {X 0,Y 641.212,Z 830.269,A -85,B 0,C 180,E1 22273.145,E2 22273.145} C_VEL
LIN {X 0,Y 639.787,Z 858.997,A -85,B 0,C 180,E1 22272.591,E2 22272.591} C_VEL
LIN {X 0,Y 638.25,Z 882.415,A -85,B 0,C 180,E1 22271.988,E2 22271.988} C_VEL
LIN {X 0,Y 636.652,Z 903.364,A -85,B 0,C 180,E1 22271.331,E2 22271.331} C_VEL
LIN {X 0,Y 634.891,Z 923.856,A -85,B 0,C 180,E1 22270.573,E2 22270.573} C_VEL
LIN {X 0,Y 632.621,Z 948.058,A -85,B 0,C 180,E1 22269.528,E2 22269.528} C_VEL
LIN {X 0,Y 629.983,Z 973.132,A -85,B 0,C 180,E1 22268.242,E2 22268.242} C_VEL
LIN {X 0,Y 627.84,Z 992.188,A -85,B 0,C 180,E1 22267.127,E2 22267.127} C_VEL
LIN {X 0,Y 625.676,Z 1010.789,A -85,B 0,C 180,E1 22265.908,E2 22265.908} C_VEL
LIN {X 0,Y 623.45,Z 1029.567,A -85,B 0,C 180,E1 22264.537,E2 22264.537} C_VEL
LIN {X 0,Y 620.866,Z 1051.281,A -85,B 0,C 180,E1 22262.759,E2 22262.759} C_VEL
LIN {X 0,Y 618.417,Z 1071.274,A -85,B 0,C 180,E1 22260.887,E2 22260.887} C_VEL
LIN {X 0,Y 616.564,Z 1087.303,A -85,B 0,C 180,E1 22259.217,E2 22259.217} C_VEL
LIN {X 0,Y 614.665,Z 1104.755,A -85,B 0,C 180,E1 22257.2,E2 22257.2} C_VEL
LIN {X 0,Y 612.799,Z 1122.416,A -85,B 0,C 180,E1 22254.876,E2 22254.876} C_VEL
LIN {X 0,Y 611.534,Z 1135.739,A -85,B 0,C 180,E1 22252.901,E2 22252.901} C_VEL
LIN {X 0,Y 610.396,Z 1149.445,A -85,B 0,C 180,E1 22250.621,E2 22250.621} C_VEL
LIN {X 0,Y 609.431,Z 1162.686,A -85,B 0,C 180,E1 22248.064,E2 22248.064} C_VEL
LIN {X 0,Y 608.873,Z 1171.901,A -85,B 0,C 180,E1 22246.015,E2 22246.015} C_VEL
LIN {X 0,Y 608.483,Z 1179.868,A -85,B 0,C 180,E1 22243.978,E2 22243.978} C_VEL
LIN {X 0,Y 608.199,Z 1187.597,A -85,B 0,C 180,E1 22241.666,E2 22241.666} C_VEL
LIN {X 0,Y 608.013,Z 1194.695,A -85,B 0,C 180,E1 22238.988,E2 22238.988} C_VEL
LIN {X 0,Y 607.943,Z 1199.393,A -85,B 0,C 180,E1 22236.611,E2 22236.611} C_VEL
LIN {X 0,Y 607.918,Z 1202.688,A -85,B 0,C 180,E1 22234.244,E2 22234.244} C_VEL
LIN {X 0,Y 607.908,Z 1204.601,A -85,B 0,C 180,E1 22231.696,E2 22231.696} C_VEL
LIN {X 0,Y 607.893,Z 1204.872,A -85,B 0,C 180,E1 22229.434,E2 22229.434} C_VEL
LIN {X 0,Y 607.912,Z 1203.998,A -85,B 0,C 180,E1 22227.266,E2 22227.266} C_VEL
LIN {X 0,Y 607.924,Z 1201.779,A -85,B 0,C 180,E1 22224.999,E2 22224.999} C_VEL
LIN {X 0,Y 607.963,Z 1197.734,A -85,B 0,C 180,E1 22222.439,E2 22222.439} C_VEL
LIN {X 0,Y 608.069,Z 1192.12,A -85,B 0,C 180,E1 22219.962,E2 22219.962} C_VEL
LIN {X 0,Y 608.252,Z 1185.486,A -85,B 0,C 180,E1 22217.66,E2 22217.66} C_VEL
LIN {X 0,Y 608.607,Z 1177.373,A -85,B 0,C 180,E1 22215.344,E2 22215.344} C_VEL
LIN {X 0,Y 609.192,Z 1166.369,A -85,B 0,C 180,E1 22212.718,E2 22212.718} C_VEL
LIN {X 0,Y 609.901,Z 1155.79,A -85,B 0,C 180,E1 22210.561,E2 22210.561} C_VEL
LIN {X 0,Y 610.802,Z 1144.281,A -85,B 0,C 180,E1 22208.488,E2 22208.488} C_VEL
LIN {X 0,Y 612.15,Z 1129.29,A -85,B 0,C 180,E1 22206.104,E2 22206.104} C_VEL
LIN {X 0,Y 613.765,Z 1112.975,A -85,B 0,C 180,E1 22203.85,E2 22203.85} C_VEL
LIN {X 0,Y 615.43,Z 1097.309,A -85,B 0,C 180,E1 22201.911,E2 22201.911} C_VEL
LIN {X 0,Y 617.805,Z 1076.845,A -85,B 0,C 180,E1 22199.672,E2 22199.672} C_VEL
LIN {X 0,Y 619.89,Z 1059.046,A -85,B 0,C 180,E1 22197.949,E2 22197.949} C_VEL
LIN {X 0,Y 621.967,Z 1041.607,A -85,B 0,C 180,E1 22196.426,E2 22196.426} C_VEL
LIN {X 0,Y 624.677,Z 1019.534,A -85,B 0,C 180,E1 22194.702,E2 22194.702} C_VEL
LIN {X 0,Y 627.359,Z 996.427,A -85,B 0,C 180,E1 22193.139,E2 22193.139} C_VEL
LIN {X 0,Y 629.492,Z 977.536,A -85,B 0,C 180,E1 22192.006,E2 22192.006} C_VEL
LIN {X 0,Y 631.517,Z 958.68,A -85,B 0,C 180,E1 22190.997,E2 22190.997} C_VEL
LIN {X 0,Y 633.559,Z 938.315,A -85,B 0,C 180,E1 22190.034,E2 22190.034} C_VEL
LIN {X 0,Y 635.905,Z 913.021,A -85,B 0,C 180,E1 22189.004,E2 22189.004} C_VEL
LIN {X 0,Y 637.951,Z 886.527,A -85,B 0,C 180,E1 22188.13,E2 22188.13} C_VEL
LIN {X 0,Y 639.427,Z 864.521,A -85,B 0,C 180,E1 22187.54,E2 22187.54} C_VEL
LIN {X 0,Y 640.646,Z 842.434,A -85,B 0,C 180,E1 22187.067,E2 22187.067} C_VEL
LIN {X 0,Y 641.747,Z 814.926,A -85,B 0,C 180,E1 22186.627,E2 22186.627} C_VEL
LIN {X 0,Y 645.325,Z 634.762,A -85,B 0,C 180,E1 22184.22,E2 22184.22} C_VEL
LIN {X 0,Y 649.272,Z 434.498,A -85,B 0,C 180,E1 22181.5,E2 22181.5} C_VEL
LIN {X 0,Y 650.04,Z 393.089,A -85,B 0,C 180,E1 22180.911,E2 22180.911} C_VEL
LIN {X 0,Y 633.194,Z 369.141,A -85,B 0,C 180,E1 22178.852,E2 22178.852} C_VEL
LIN {X 0,Y 622.033,Z 353.85,A -85,B 0,C 180,E1 22177.36,E2 22177.36} C_VEL
LIN {X 0,Y 616.179,Z 342.334,A -85,B 0,C 180,E1 22175.631,E2 22175.631} C_VEL
LIN {X 0,Y 611.628,Z 333.556,A -85,B 0,C 180,E1 22174.22,E2 22174.22} C_VEL
LIN {X 0,Y 609.286,Z 329.683,A -85,B 0,C 180,E1 22173.523,E2 22173.523} C_VEL
LIN {X 0,Y 609.036,Z 328.555,A -85,B 0,C 180,E1 22173.317,E2 22173.317} C_VEL
LIN {X 0,Y 609.079,Z 328.362,A -85,B 0,C 180,E1 22170.591,E2 22170.591} C_VEL
LIN {X 0,Y 609.009,Z 328.332,A -85,B 0,C 180,E1 22167.475,E2 22167.475} C_VEL
LIN {X 0,Y 609.075,Z 328.33,A -85,B 0,C 180,E1 22164.437,E2 22164.437} C_VEL
LIN {X 0,Y 609.02,Z 328.362,A -85,B 0,C 180,E1 22161.376,E2 22161.376} C_VEL
LIN {X 0,Y 609.073,Z 328.315,A -85,B 0,C 180,E1 22158.274,E2 22158.274} C_VEL
LIN {X 0,Y 609.03,Z 328.366,A -85,B 0,C 180,E1 22155.126,E2 22155.126} C_VEL
LIN {X 0,Y 609.07,Z 328.313,A -85,B 0,C 180,E1 22152.034,E2 22152.034} C_VEL
LIN {X 0,Y 609.042,Z 328.366,A -85,B 0,C 180,E1 22148.878,E2 22148.878} C_VEL
LIN {X 0,Y 609.066,Z 328.315,A -85,B 0,C 180,E1 22145.653,E2 22145.653} C_VEL
LIN {X 0,Y 609.065,Z 328.361,A -85,B 0,C 180,E1 22142.446,E2 22142.446} C_VEL
LIN {X 0,Y 609.05,Z 328.317,A -85,B 0,C 180,E1 22139.153,E2 22139.153} C_VEL
LIN {X 0,Y 609.066,Z 328.355,A -85,B 0,C 180,E1 22136.046,E2 22136.046} C_VEL
LIN {X 0,Y 609.049,Z 328.315,A -85,B 0,C 180,E1 22132.832,E2 22132.832} C_VEL
LIN {X 0,Y 609.059,Z 328.353,A -85,B 0,C 180,E1 22129.692,E2 22129.692} C_VEL
LIN {X 0,Y 609.058,Z 328.32,A -85,B 0,C 180,E1 22126.519,E2 22126.519} C_VEL
LIN {X 0,Y 609.056,Z 328.353,A -85,B 0,C 180,E1 22123.402,E2 22123.402} C_VEL
LIN {X 0,Y 609.069,Z 328.337,A -85,B 0,C 180,E1 22120.134,E2 22120.134} C_VEL
LIN {X 0,Y 609.068,Z 328.325,A -85,B 0,C 180,E1 22116.898,E2 22116.898} C_VEL
LIN {X 0,Y 609.052,Z 328.368,A -85,B 0,C 180,E1 22113.685,E2 22113.685} C_VEL
LIN {X 0,Y 609.072,Z 328.319,A -85,B 0,C 180,E1 22110.603,E2 22110.603} C_VEL
LIN {X 0,Y 609.039,Z 328.333,A -85,B 0,C 180,E1 22107.53,E2 22107.53} C_VEL
LIN {X 0,Y 609.064,Z 328.567,A -85,B 0,C 180,E1 22105.023,E2 22105.023} C_VEL
LIN {X 0,Y 610.421,Z 331.906,A -85,B 0,C 180,E1 22104.444,E2 22104.444} C_VEL
LIN {X 0,Y 611.694,Z 333.94,A -85,B 0,C 180,E1 22104.067,E2 22104.067} C_VEL
LIN {X 0,Y 617.054,Z 344.508,A -85,B 0,C 180,E1 22102.345,E2 22102.345} C_VEL
LIN {X 0,Y 623.016,Z 356.356,A -85,B 0,C 180,E1 22100.53,E2 22100.53} C_VEL
LIN {X 0,Y 630.438,Z 372.014,A -85,B 0,C 180,E1 22098.332,E2 22098.332} C_VEL
LIN {X 0,Y 637.134,Z 387.123,A -85,B 0,C 180,E1 22096.391,E2 22096.391} C_VEL
LIN {X 0,Y 636.784,Z 393.785,A -85,B 0,C 180,E1 22095.933,E2 22095.933} C_VEL
LIN {X 0,Y 644.938,Z 432.416,A -85,B 0,C 180,E1 22094.527,E2 22094.527} C_VEL
LIN {X 0,Y 644.124,Z 471.524,A -85,B 0,C 180,E1 22093.998,E2 22093.998} C_VEL
LIN {X 0,Y 643.264,Z 479.229,A -85,B 0,C 180,E1 22093.959,E2 22093.959} C_VEL
LIN {X 0,Y 638.466,Z 499.878,A -85,B 0,C 180,E1 22094.089,E2 22094.089} C_VEL
LIN {X 0,Y 637.787,Z 506.491,A -85,B 0,C 180,E1 22094.05,E2 22094.05} C_VEL
LIN {X 0,Y 633.028,Z 726.38,A -85,B 0,C 180,E1 22091.113,E2 22091.113} C_VEL
LIN {X 0,Y 630.558,Z 830.881,A -85,B 0,C 180,E1 22089.704,E2 22089.704} C_VEL
LIN {X 0,Y 629.242,Z 857.649,A -85,B 0,C 180,E1 22089.197,E2 22089.197} C_VEL
LIN {X 0,Y 627.707,Z 880.277,A -85,B 0,C 180,E1 22088.611,E2 22088.611} C_VEL
LIN {X 0,Y 626.03,Z 901.08,A -85,B 0,C 180,E1 22087.946,E2 22087.946} C_VEL
LIN {X 0,Y 623.836,Z 925.448,A -85,B 0,C 180,E1 22087.002,E2 22087.002} C_VEL
LIN {X 0,Y 621.478,Z 947.647,A -85,B 0,C 180,E1 22085.961,E2 22085.961} C_VEL
LIN {X 0,Y 619.398,Z 966.145,A -85,B 0,C 180,E1 22084.965,E2 22084.965} C_VEL
LIN {X 0,Y 617.181,Z 984.966,A -85,B 0,C 180,E1 22083.814,E2 22083.814} C_VEL
LIN {X 0,Y 614.289,Z 1009.668,A -85,B 0,C 180,E1 22082.103,E2 22082.103} C_VEL
LIN {X 0,Y 612.223,Z 1027.586,A -85,B 0,C 180,E1 22080.689,E2 22080.689} C_VEL
LIN {X 0,Y 610.031,Z 1046.99,A -85,B 0,C 180,E1 22078.97,E2 22078.97} C_VEL
LIN {X 0,Y 607.848,Z 1065.799,A -85,B 0,C 180,E1 22077.054,E2 22077.054} C_VEL
LIN {X 0,Y 606.191,Z 1081.225,A -85,B 0,C 180,E1 22075.291,E2 22075.291} C_VEL
LIN {X 0,Y 604.443,Z 1098.284,A -85,B 0,C 180,E1 22073.082,E2 22073.082} C_VEL
LIN {X 0,Y 603.186,Z 1111.771,A -85,B 0,C 180,E1 22071.083,E2 22071.083} C_VEL
LIN {X 0,Y 602.075,Z 1125.369,A -85,B 0,C 180,E1 22068.804,E2 22068.804} C_VEL
LIN {X 0,Y 601.246,Z 1136.938,A -85,B 0,C 180,E1 22066.522,E2 22066.522} C_VEL
LIN {X 0,Y 600.717,Z 1146.004,A -85,B 0,C 180,E1 22064.458,E2 22064.458} C_VEL
LIN {X 0,Y 600.317,Z 1155.109,A -85,B 0,C 180,E1 22062.017,E2 22062.017} C_VEL
LIN {X 0,Y 600.077,Z 1161.767,A -85,B 0,C 180,E1 22059.786,E2 22059.786} C_VEL
LIN {X 0,Y 599.991,Z 1166.438,A -85,B 0,C 180,E1 22057.854,E2 22057.854} C_VEL
LIN {X 0,Y 599.918,Z 1170.233,A -85,B 0,C 180,E1 22055.835,E2 22055.835} C_VEL
LIN {X 0,Y 599.9,Z 1173.356,A -85,B 0,C 180,E1 22053.44,E2 22053.44} C_VEL
LIN {X 0,Y 599.91,Z 1174.746,A -85,B 0,C 180,E1 22051.051,E2 22051.051} C_VEL
LIN {X 0,Y 599.907,Z 1174.791,A -85,B 0,C 180,E1 22049.045,E2 22049.045} C_VEL
LIN {X 0,Y 599.906,Z 1173.767,A -85,B 0,C 180,E1 22047.039,E2 22047.039} C_VEL
LIN {X 0,Y 599.92,Z 1171.017,A -85,B 0,C 180,E1 22044.549,E2 22044.549} C_VEL
LIN {X 0,Y 599.974,Z 1166.838,A -85,B 0,C 180,E1 22042.242,E2 22042.242} C_VEL
LIN {X 0,Y 600.068,Z 1162.259,A -85,B 0,C 180,E1 22040.312,E2 22040.312} C_VEL
LIN {X 0,Y 600.266,Z 1156.306,A -85,B 0,C 180,E1 22038.275,E2 22038.275} C_VEL
LIN {X 0,Y 600.655,Z 1147.19,A -85,B 0,C 180,E1 22035.738,E2 22035.738} C_VEL
LIN {X 0,Y 601.193,Z 1137.814,A -85,B 0,C 180,E1 22033.577,E2 22033.577} C_VEL
LIN {X 0,Y 601.904,Z 1127.453,A -85,B 0,C 180,E1 22031.501,E2 22031.501} C_VEL
LIN {X 0,Y 603.022,Z 1113.608,A -85,B 0,C 180,E1 22029.115,E2 22029.115} C_VEL
LIN {X 0,Y 604.187,Z 1100.829,A -85,B 0,C 180,E1 22027.191,E2 22027.191} C_VEL
LIN {X 0,Y 605.787,Z 1085.284,A -85,B 0,C 180,E1 22025.11,E2 22025.11} C_VEL
LIN {X 0,Y 607.611,Z 1067.984,A -85,B 0,C 180,E1 22023.094,E2 22023.094} C_VEL
LIN {X 0,Y 609.357,Z 1052.455,A -85,B 0,C 180,E1 22021.478,E2 22021.478} C_VEL
LIN {X 0,Y 611.671,Z 1032.867,A -85,B 0,C 180,E1 22019.662,E2 22019.662} C_VEL
LIN {X 0,Y 613.938,Z 1012.778,A -85,B 0,C 180,E1 22018.042,E2 22018.042} C_VEL
LIN {X 0,Y 616.294,Z 992.316,A -85,B 0,C 180,E1 22016.578,E2 22016.578} C_VEL
LIN {X 0,Y 619.039,Z 969.277,A -85,B 0,C 180,E1 22015.126,E2 22015.126} C_VEL
LIN {X 0,Y 621.195,Z 950.165,A -85,B 0,C 180,E1 22014.077,E2 22014.077} C_VEL
LIN {X 0,Y 623.282,Z 930.437,A -85,B 0,C 180,E1 22013.132,E2 22013.132} C_VEL
LIN {X 0,Y 625.665,Z 905.958,A -85,B 0,C 180,E1 22012.137,E2 22012.137} C_VEL
LIN {X 0,Y 627.501,Z 883.206,A -85,B 0,C 180,E1 22011.386,E2 22011.386} C_VEL
LIN {X 0,Y 628.882,Z 863.451,A -85,B 0,C 180,E1 22010.854,E2 22010.854} C_VEL
LIN {X 0,Y 630.016,Z 843.6,A -85,B 0,C 180,E1 22010.427,E2 22010.427} C_VEL
LIN {X 0,Y 631.051,Z 816.409,A -85,B 0,C 180,E1 22009.994,E2 22009.994} C_VEL
LIN {X 0,Y 635.69,Z 604.42,A -85,B 0,C 180,E1 22007.172,E2 22007.172} C_VEL
LIN {X 0,Y 639.351,Z 433.904,A -85,B 0,C 180,E1 22004.87,E2 22004.87} C_VEL
LIN {X 0,Y 630.746,Z 392.35,A -85,B 0,C 180,E1 22003.313,E2 22003.313} C_VEL
LIN {X 0,Y 630.588,Z 390.672,A -85,B 0,C 180,E1 22003.165,E2 22003.165} C_VEL
LIN {X 0,Y 622.354,Z 372.131,A -85,B 0,C 180,E1 22000.715,E2 22000.715} C_VEL
LIN {X 0,Y 614.608,Z 356.115,A -85,B 0,C 180,E1 21998.359,E2 21998.359} C_VEL
LIN {X 0,Y 609.819,Z 346.725,A -85,B 0,C 180,E1 21996.857,E2 21996.857} C_VEL
LIN {X 0,Y 605.464,Z 338.232,A -85,B 0,C 180,E1 21995.427,E2 21995.427} C_VEL
LIN {X 0,Y 603.178,Z 333.831,A -85,B 0,C 180,E1 21994.652,E2 21994.652} C_VEL
LIN {X 0,Y 601.432,Z 330.744,A -85,B 0,C 180,E1 21994.075,E2 21994.075} C_VEL
LIN {X 0,Y 601.151,Z 329.432,A -85,B 0,C 180,E1 21993.805,E2 21993.805} C_VEL
LIN {X 0,Y 601.092,Z 329.345,A -85,B 0,C 180,E1 21990.599,E2 21990.599} C_VEL
LIN {X 0,Y 601.135,Z 329.324,A -85,B 0,C 180,E1 21987.435,E2 21987.435} C_VEL
LIN {X 0,Y 601.103,Z 329.309,A -85,B 0,C 180,E1 21984.259,E2 21984.259} C_VEL
LIN {X 0,Y 601.128,Z 329.351,A -85,B 0,C 180,E1 21980.954,E2 21980.954} C_VEL
LIN {X 0,Y 601.128,Z 329.306,A -85,B 0,C 180,E1 21977.722,E2 21977.722} C_VEL
LIN {X 0,Y 601.115,Z 329.34,A -85,B 0,C 180,E1 21974.516,E2 21974.516} C_VEL
LIN {X 0,Y 601.119,Z 329.314,A -85,B 0,C 180,E1 21971.32,E2 21971.32} C_VEL
LIN {X 0,Y 601.117,Z 329.326,A -85,B 0,C 180,E1 21968.128,E2 21968.128} C_VEL
LIN {X 0,Y 601.116,Z 329.321,A -85,B 0,C 180,E1 21964.962,E2 21964.962} C_VEL
LIN {X 0,Y 601.13,Z 329.321,A -85,B 0,C 180,E1 21961.716,E2 21961.716} C_VEL
LIN {X 0,Y 601.133,Z 329.333,A -85,B 0,C 180,E1 21958.38,E2 21958.38} C_VEL
LIN {X 0,Y 601.104,Z 329.32,A -85,B 0,C 180,E1 21955.133,E2 21955.133} C_VEL
LIN {X 0,Y 601.132,Z 329.334,A -85,B 0,C 180,E1 21951.968,E2 21951.968} C_VEL
LIN {X 0,Y 601.094,Z 329.316,A -85,B 0,C 180,E1 21948.874,E2 21948.874} C_VEL
LIN {X 0,Y 601.137,Z 329.341,A -85,B 0,C 180,E1 21945.65,E2 21945.65} C_VEL
LIN {X 0,Y 601.087,Z 329.309,A -85,B 0,C 180,E1 21942.577,E2 21942.577} C_VEL
LIN {X 0,Y 601.129,Z 329.355,A -85,B 0,C 180,E1 21939.352,E2 21939.352} C_VEL
LIN {X 0,Y 601.08,Z 329.31,A -85,B 0,C 180,E1 21936.365,E2 21936.365} C_VEL
LIN {X 0,Y 601.104,Z 329.327,A -85,B 0,C 180,E1 21933.099,E2 21933.099} C_VEL
LIN {X 0,Y 601.078,Z 329.341,A -85,B 0,C 180,E1 21930.173,E2 21930.173} C_VEL
LIN {X 0,Y 601.148,Z 329.551,A -85,B 0,C 180,E1 21927.695,E2 21927.695} C_VEL
LIN {X 0,Y 602.75,Z 333.271,A -85,B 0,C 180,E1 21927.036,E2 21927.036} C_VEL
LIN {X 0,Y 603.953,Z 335.367,A -85,B 0,C 180,E1 21926.657,E2 21926.657} C_VEL
LIN {X 0,Y 606.924,Z 340.933,A -85,B 0,C 180,E1 21925.706,E2 21925.706} C_VEL
LIN {X 0,Y 609.337,Z 345.553,A -85,B 0,C 180,E1 21924.947,E2 21924.947} C_VEL
LIN {X 0,Y 613.913,Z 354.242,A -85,B 0,C 180,E1 21923.569,E2 21923.569} C_VEL
LIN {X 0,Y 624.883,Z 369.234,A -85,B 0,C 180,E1 21922.03,E2 21922.03} C_VEL
LIN {X 0,Y 634.941,Z 383.376,A -85,B 0,C 180,E1 21920.723,E2 21920.723} C_VEL
LIN {X 0,Y 644.593,Z 397.345,A -85,B 0,C 180,E1 21919.539,E2 21919.539} C_VEL
LIN {X 0,Y 640.17,Z 597.971,A -85,B 0,C 180,E1 21916.765,E2 21916.765} C_VEL
LIN {X 0,Y 635.81,Z 818.463,A -85,B 0,C 180,E1 21913.817,E2 21913.817} C_VEL
LIN {X 0,Y 634.738,Z 843.126,A -85,B 0,C 180,E1 21913.414,E2 21913.414} C_VEL
LIN {X 0,Y 633.486,Z 864.616,A -85,B 0,C 180,E1 21912.95,E2 21912.95} C_VEL
LIN {X 0,Y 631.957,Z 886.323,A -85,B 0,C 180,E1 21912.365,E2 21912.365} C_VEL
LIN {X 0,Y 629.909,Z 911.495,A -85,B 0,C 180,E1 21911.537,E2 21911.537} C_VEL
LIN {X 0,Y 627.434,Z 937.187,A -85,B 0,C 180,E1 21910.495,E2 21910.495} C_VEL
LIN {X 0,Y 625.261,Z 957.675,A -85,B 0,C 180,E1 21909.528,E2 21909.528} C_VEL
LIN {X 0,Y 623.097,Z 976.73,A -85,B 0,C 180,E1 21908.507,E2 21908.507} C_VEL
LIN {X 0,Y 620.862,Z 995.431,A -85,B 0,C 180,E1 21907.383,E2 21907.383} C_VEL
LIN {X 0,Y 618.34,Z 1015.929,A -85,B 0,C 180,E1 21906,E2 21906} C_VEL
LIN {X 0,Y 615.313,Z 1039.359,A -85,B 0,C 180,E1 21904.194,E2 21904.194} C_VEL
LIN {X 0,Y 612.992,Z 1057.385,A -85,B 0,C 180,E1 21902.622,E2 21902.622} C_VEL
LIN {X 0,Y 610.906,Z 1073.807,A -85,B 0,C 180,E1 21901.035,E2 21901.035} C_VEL
LIN {X 0,Y 608.726,Z 1091.946,A -85,B 0,C 180,E1 21899.089,E2 21899.089} C_VEL
LIN {X 0,Y 606.521,Z 1110.305,A -85,B 0,C 180,E1 21896.853,E2 21896.853} C_VEL
LIN {X 0,Y 604.943,Z 1124.923,A -85,B 0,C 180,E1 21894.848,E2 21894.848} C_VEL
LIN {X 0,Y 603.439,Z 1140.181,A -85,B 0,C 180,E1 21892.504,E2 21892.504} C_VEL
LIN {X 0,Y 602.197,Z 1154.242,A -85,B 0,C 180,E1 21890.001,E2 21890.001} C_VEL
LIN {X 0,Y 601.435,Z 1164.532,A -85,B 0,C 180,E1 21887.912,E2 21887.912} C_VEL
LIN {X 0,Y 600.808,Z 1174.331,A -85,B 0,C 180,E1 21885.64,E2 21885.64} C_VEL
LIN {X 0,Y 600.353,Z 1184.273,A -85,B 0,C 180,E1 21882.895,E2 21882.895} C_VEL
LIN {X 0,Y 600.109,Z 1191.1,A -85,B 0,C 180,E1 21880.561,E2 21880.561} C_VEL
LIN {X 0,Y 599.988,Z 1196.552,A -85,B 0,C 180,E1 21878.24,E2 21878.24} C_VEL
LIN {X 0,Y 599.932,Z 1201.053,A -85,B 0,C 180,E1 21875.643,E2 21875.643} C_VEL
LIN {X 0,Y 599.917,Z 1203.724,A -85,B 0,C 180,E1 21873.153,E2 21873.153} C_VEL
LIN {X 0,Y 599.912,Z 1204.759,A -85,B 0,C 180,E1 21871.05,E2 21871.05} C_VEL
LIN {X 0,Y 599.909,Z 1204.782,A -85,B 0,C 180,E1 21869.045,E2 21869.045} C_VEL
LIN {X 0,Y 599.918,Z 1203.791,A -85,B 0,C 180,E1 21866.943,E2 21866.943} C_VEL
LIN {X 0,Y 599.928,Z 1201.177,A -85,B 0,C 180,E1 21864.453,E2 21864.453} C_VEL
LIN {X 0,Y 599.985,Z 1196.757,A -85,B 0,C 180,E1 21861.856,E2 21861.856} C_VEL
LIN {X 0,Y 600.105,Z 1191.354,A -85,B 0,C 180,E1 21859.536,E2 21859.536} C_VEL
LIN {X 0,Y 600.338,Z 1184.574,A -85,B 0,C 180,E1 21857.202,E2 21857.202} C_VEL
LIN {X 0,Y 600.788,Z 1174.733,A -85,B 0,C 180,E1 21854.458,E2 21854.458} C_VEL
LIN {X 0,Y 601.405,Z 1164.992,A -85,B 0,C 180,E1 21852.187,E2 21852.187} C_VEL
LIN {X 0,Y 602.16,Z 1154.759,A -85,B 0,C 180,E1 21850.099,E2 21850.099} C_VEL
LIN {X 0,Y 603.269,Z 1141.954,A -85,B 0,C 180,E1 21847.796,E2 21847.796} C_VEL
LIN {X 0,Y 604.785,Z 1126.485,A -85,B 0,C 180,E1 21845.378,E2 21845.378} C_VEL
LIN {X 0,Y 606.34,Z 1111.842,A -85,B 0,C 180,E1 21843.35,E2 21843.35} C_VEL
LIN {X 0,Y 608.291,Z 1095.436,A -85,B 0,C 180,E1 21841.316,E2 21841.316} C_VEL
LIN {X 0,Y 610.669,Z 1075.83,A -85,B 0,C 180,E1 21839.17,E2 21839.17} C_VEL
LIN {X 0,Y 612.802,Z 1058.913,A -85,B 0,C 180,E1 21837.52,E2 21837.52} C_VEL
LIN {X 0,Y 615.006,Z 1041.605,A -85,B 0,C 180,E1 21835.994,E2 21835.994} C_VEL
LIN {X 0,Y 617.905,Z 1019.533,A -85,B 0,C 180,E1 21834.256,E2 21834.256} C_VEL
LIN {X 0,Y 620.669,Z 997.039,A -85,B 0,C 180,E1 21832.719,E2 21832.719} C_VEL
LIN {X 0,Y 622.994,Z 977.624,A -85,B 0,C 180,E1 21831.543,E2 21831.543} C_VEL
LIN {X 0,Y 625.15,Z 958.676,A -85,B 0,C 180,E1 21830.523,E2 21830.523} C_VEL
LIN {X 0,Y 627.188,Z 939.443,A -85,B 0,C 180,E1 21829.605,E2 21829.605} C_VEL
LIN {X 0,Y 629.337,Z 917.421,A -85,B 0,C 180,E1 21828.689,E2 21828.689} C_VEL
LIN {X 0,Y 631.747,Z 889.222,A -85,B 0,C 180,E1 21827.72,E2 21827.72} C_VEL
LIN {X 0,Y 633.402,Z 865.97,A -85,B 0,C 180,E1 21827.083,E2 21827.083} C_VEL
LIN {X 0,Y 634.662,Z 844.614,A -85,B 0,C 180,E1 21826.615,E2 21826.615} C_VEL
LIN {X 0,Y 635.665,Z 822.269,A -85,B 0,C 180,E1 21826.24,E2 21826.24} C_VEL
LIN {X 0,Y 638.411,Z 686.235,A -85,B 0,C 180,E1 21824.423,E2 21824.423} C_VEL
LIN {X 0,Y 642.726,Z 477.791,A -85,B 0,C 180,E1 21821.589,E2 21821.589} C_VEL
LIN {X 0,Y 644.482,Z 397.048,A -85,B 0,C 180,E1 21820.446,E2 21820.446} C_VEL
LIN {X 0,Y 628.735,Z 374.539,A -85,B 0,C 180,E1 21818.478,E2 21818.478} C_VEL
LIN {X 0,Y 616.318,Z 357.556,A -85,B 0,C 180,E1 21816.803,E2 21816.803} C_VEL
LIN {X 0,Y 613.941,Z 354.28,A -85,B 0,C 180,E1 21816.434,E2 21816.434} C_VEL
LIN {X 0,Y 610.129,Z 347.058,A -85,B 0,C 180,E1 21815.301,E2 21815.301} C_VEL
LIN {X 0,Y 605.741,Z 338.594,A -85,B 0,C 180,E1 21813.913,E2 21813.913} C_VEL
LIN {X 0,Y 603.686,Z 334.591,A -85,B 0,C 180,E1 21813.235,E2 21813.235} C_VEL
LIN {X 0,Y 601.367,Z 330.486,A -85,B 0,C 180,E1 21812.483,E2 21812.483} C_VEL
LIN {X 0,Y 601.139,Z 329.524,A -85,B 0,C 180,E1 21812.271,E2 21812.271} C_VEL
LIN {X 0,Y 601.072,Z 329.325,A -85,B 0,C 180,E1 21809.28,E2 21809.28} C_VEL
LIN {X 0,Y 601.115,Z 329.353,A -85,B 0,C 180,E1 21806.075,E2 21806.075} C_VEL
LIN {X 0,Y 601.087,Z 329.309,A -85,B 0,C 180,E1 21803.012,E2 21803.012} C_VEL
LIN {X 0,Y 601.099,Z 329.34,A -85,B 0,C 180,E1 21799.696,E2 21799.696} C_VEL
LIN {X 0,Y 601.119,Z 329.322,A -85,B 0,C 180,E1 21796.625,E2 21796.625} C_VEL
LIN {X 0,Y 601.098,Z 329.323,A -85,B 0,C 180,E1 21793.467,E2 21793.467} C_VEL
LIN {X 0,Y 601.131,Z 329.33,A -85,B 0,C 180,E1 21790.349,E2 21790.349} C_VEL
LIN {X 0,Y 601.097,Z 329.315,A -85,B 0,C 180,E1 21787.167,E2 21787.167} C_VEL
LIN {X 0,Y 601.13,Z 329.337,A -85,B 0,C 180,E1 21784.006,E2 21784.006} C_VEL
LIN {X 0,Y 601.103,Z 329.313,A -85,B 0,C 180,E1 21780.858,E2 21780.858} C_VEL
LIN {X 0,Y 601.127,Z 329.337,A -85,B 0,C 180,E1 21777.712,E2 21777.712} C_VEL
LIN {X 0,Y 601.119,Z 329.305,A -85,B 0,C 180,E1 21774.464,E2 21774.464} C_VEL
LIN {X 0,Y 601.129,Z 329.343,A -85,B 0,C 180,E1 21771.101,E2 21771.101} C_VEL
LIN {X 0,Y 601.116,Z 329.3,A -85,B 0,C 180,E1 21767.902,E2 21767.902} C_VEL
LIN {X 0,Y 601.125,Z 329.349,A -85,B 0,C 180,E1 21764.74,E2 21764.74} C_VEL
LIN {X 0,Y 601.108,Z 329.303,A -85,B 0,C 180,E1 21761.576,E2 21761.576} C_VEL
LIN {X 0,Y 601.131,Z 329.348,A -85,B 0,C 180,E1 21758.33,E2 21758.33} C_VEL
LIN {X 0,Y 601.109,Z 329.318,A -85,B 0,C 180,E1 21755.112,E2 21755.112} C_VEL
LIN {X 0,Y 601.118,Z 329.311,A -85,B 0,C 180,E1 21751.834,E2 21751.834} C_VEL
LIN {X 0,Y 601.135,Z 329.35,A -85,B 0,C 180,E1 21748.626,E2 21748.626} C_VEL
LIN {X 0,Y 601.163,Z 329.53,A -85,B 0,C 180,E1 21746.042,E2 21746.042} C_VEL
LIN {X 0,Y 602.543,Z 333.016,A -85,B 0,C 180,E1 21745.421,E2 21745.421} C_VEL
LIN {X 0,Y 603.786,Z 334.977,A -85,B 0,C 180,E1 21745.041,E2 21745.041} C_VEL
LIN {X 0,Y 606.385,Z 339.972,A -85,B 0,C 180,E1 21744.17,E2 21744.17} C_VEL
LIN {X 0,Y 612.724,Z 352.161,A -85,B 0,C 180,E1 21742.151,E2 21742.151} C_VEL
LIN {X 0,Y 621.148,Z 369.548,A -85,B 0,C 180,E1 21739.554,E2 21739.554} C_VEL
LIN {X 0,Y 629.216,Z 387.5,A -85,B 0,C 180,E1 21737.145,E2 21737.145} C_VEL
LIN {X 0,Y 630.793,Z 391.475,A -85,B 0,C 180,E1 21736.657,E2 21736.657} C_VEL
LIN {X 0,Y 631.085,Z 394.521,A -85,B 0,C 180,E1 21736.502,E2 21736.502} C_VEL
LIN {X 0,Y 639.419,Z 434.337,A -85,B 0,C 180,E1 21735.025,E2 21735.025} C_VEL
LIN {X 0,Y 637.787,Z 506.491,A -85,B 0,C 180,E1 21734.05,E2 21734.05} C_VEL
LIN {X 0,Y 636.911,Z 514.199,A -85,B 0,C 180,E1 21734.014,E2 21734.014} C_VEL
LIN {X 0,Y 632.116,Z 534.847,A -85,B 0,C 180,E1 21734.148,E2 21734.148} C_VEL
LIN {X 0,Y 631.458,Z 541.457,A -85,B 0,C 180,E1 21734.107,E2 21734.107} C_VEL
LIN {X 0,Y 626.725,Z 752.525,A -85,B 0,C 180,E1 21731.279,E2 21731.279} C_VEL
LIN {X 0,Y 624.782,Z 831.099,A -85,B 0,C 180,E1 21730.211,E2 21730.211} C_VEL
LIN {X 0,Y 623.42,Z 857.609,A -85,B 0,C 180,E1 21729.709,E2 21729.709} C_VEL
LIN {X 0,Y 621.771,Z 880.667,A -85,B 0,C 180,E1 21729.108,E2 21729.108} C_VEL
LIN {X 0,Y 620.008,Z 901.453,A -85,B 0,C 180,E1 21728.44,E2 21728.44} C_VEL
LIN {X 0,Y 617.694,Z 925.793,A -85,B 0,C 180,E1 21727.491,E2 21727.491} C_VEL
LIN {X 0,Y 615.163,Z 948.201,A -85,B 0,C 180,E1 21726.43,E2 21726.43} C_VEL
LIN {X 0,Y 612.983,Z 966.336,A -85,B 0,C 180,E1 21725.442,E2 21725.442} C_VEL
LIN {X 0,Y 610.632,Z 985.155,A -85,B 0,C 180,E1 21724.283,E2 21724.283} C_VEL
LIN {X 0,Y 607.64,Z 1008.023,A -85,B 0,C 180,E1 21722.665,E2 21722.665} C_VEL
LIN {X 0,Y 604.493,Z 1033.066,A -85,B 0,C 180,E1 21720.628,E2 21720.628} C_VEL
LIN {X 0,Y 602.038,Z 1052.616,A -85,B 0,C 180,E1 21718.793,E2 21718.793} C_VEL
LIN {X 0,Y 600.172,Z 1068.117,A -85,B 0,C 180,E1 21717.16,E2 21717.16} C_VEL
LIN {X 0,Y 598.232,Z 1085.398,A -85,B 0,C 180,E1 21715.121,E2 21715.121} C_VEL
LIN {X 0,Y 596.499,Z 1101.089,A -85,B 0,C 180,E1 21712.99,E2 21712.99} C_VEL
LIN {X 0,Y 595.196,Z 1114.572,A -85,B 0,C 180,E1 21710.925,E2 21710.925} C_VEL
LIN {X 0,Y 594.025,Z 1128.024,A -85,B 0,C 180,E1 21708.55,E2 21708.55} C_VEL
LIN {X 0,Y 593.27,Z 1138.315,A -85,B 0,C 180,E1 21706.448,E2 21706.448} C_VEL
LIN {X 0,Y 592.665,Z 1148.482,A -85,B 0,C 180,E1 21704.048,E2 21704.048} C_VEL
LIN {X 0,Y 592.285,Z 1156.634,A -85,B 0,C 180,E1 21701.688,E2 21701.688} C_VEL
LIN {X 0,Y 592.08,Z 1162.532,A -85,B 0,C 180,E1 21699.624,E2 21699.624} C_VEL
LIN {X 0,Y 591.971,Z 1167.474,A -85,B 0,C 180,E1 21697.473,E2 21697.473} C_VEL
LIN {X 0,Y 591.913,Z 1171.667,A -85,B 0,C 180,E1 21694.942,E2 21694.942} C_VEL
LIN {X 0,Y 591.904,Z 1173.904,A -85,B 0,C 180,E1 21692.711,E2 21692.711} C_VEL
LIN {X 0,Y 591.895,Z 1174.836,A -85,B 0,C 180,E1 21690.678,E2 21690.678} C_VEL
LIN {X 0,Y 591.907,Z 1174.656,A -85,B 0,C 180,E1 21688.451,E2 21688.451} C_VEL
LIN {X 0,Y 591.915,Z 1172.797,A -85,B 0,C 180,E1 21685.932,E2 21685.932} C_VEL
LIN {X 0,Y 591.942,Z 1169.901,A -85,B 0,C 180,E1 21683.794,E2 21683.794} C_VEL
LIN {X 0,Y 592.01,Z 1166.011,A -85,B 0,C 180,E1 21681.746,E2 21681.746} C_VEL
LIN {X 0,Y 592.169,Z 1159.942,A -85,B 0,C 180,E1 21679.296,E2 21679.296} C_VEL
LIN {X 0,Y 592.472,Z 1152.319,A -85,B 0,C 180,E1 21676.93,E2 21676.93} C_VEL
LIN {X 0,Y 592.896,Z 1144.347,A -85,B 0,C 180,E1 21674.847,E2 21674.847} C_VEL
LIN {X 0,Y 593.62,Z 1133.544,A -85,B 0,C 180,E1 21672.434,E2 21672.434} C_VEL
LIN {X 0,Y 594.577,Z 1121.345,A -85,B 0,C 180,E1 21670.142,E2 21670.142} C_VEL
LIN {X 0,Y 595.69,Z 1109.152,A -85,B 0,C 180,E1 21668.122,E2 21668.122} C_VEL
LIN {X 0,Y 597.363,Z 1093.004,A -85,B 0,C 180,E1 21665.79,E2 21665.79} C_VEL
LIN {X 0,Y 598.962,Z 1078.565,A -85,B 0,C 180,E1 21663.958,E2 21663.958} C_VEL
LIN {X 0,Y 600.886,Z 1062.41,A -85,B 0,C 180,E1 21662.123,E2 21662.123} C_VEL
LIN {X 0,Y 603.227,Z 1042.934,A -85,B 0,C 180,E1 21660.181,E2 21660.181} C_VEL
LIN {X 0,Y 605.371,Z 1025.464,A -85,B 0,C 180,E1 21658.642,E2 21658.642} C_VEL
LIN {X 0,Y 608.511,Z 1001.524,A -85,B 0,C 180,E1 21656.76,E2 21656.76} C_VEL
LIN {X 0,Y 610.956,Z 982.485,A -85,B 0,C 180,E1 21655.454,E2 21655.454} C_VEL
LIN {X 0,Y 613.345,Z 963.367,A -85,B 0,C 180,E1 21654.295,E2 21654.295} C_VEL
LIN {X 0,Y 616.157,Z 939.473,A -85,B 0,C 180,E1 21653.042,E2 21653.042} C_VEL
LIN {X 0,Y 618.427,Z 917.893,A -85,B 0,C 180,E1 21652.093,E2 21652.093} C_VEL
LIN {X 0,Y 620.377,Z 897.226,A -85,B 0,C 180,E1 21651.322,E2 21651.322} C_VEL
LIN {X 0,Y 622.513,Z 871.524,A -85,B 0,C 180,E1 21650.543,E2 21650.543} C_VEL
LIN {X 0,Y 623.954,Z 848.461,A -85,B 0,C 180,E1 21650.011,E2 21650.011} C_VEL
LIN {X 0,Y 624.96,Z 826.62,A -85,B 0,C 180,E1 21649.631,E2 21649.631} C_VEL
LIN {X 0,Y 628.949,Z 655.373,A -85,B 0,C 180,E1 21647.332,E2 21647.332} C_VEL
LIN {X 0,Y 633.911,Z 435.972,A -85,B 0,C 180,E1 21644.368,E2 21644.368} C_VEL
LIN {X 0,Y 625.579,Z 395.978,A -85,B 0,C 180,E1 21642.851,E2 21642.851} C_VEL
LIN {X 0,Y 622.72,Z 391.165,A -85,B 0,C 180,E1 21642.407,E2 21642.407} C_VEL
LIN {X 0,Y 614.728,Z 373.458,A -85,B 0,C 180,E1 21639.978,E2 21639.978} C_VEL
LIN {X 0,Y 608.496,Z 360.633,A -85,B 0,C 180,E1 21638.04,E2 21638.04} C_VEL
LIN {X 0,Y 604.281,Z 352.206,A -85,B 0,C 180,E1 21636.68,E2 21636.68} C_VEL
LIN {X 0,Y 600.028,Z 343.899,A -85,B 0,C 180,E1 21635.262,E2 21635.262} C_VEL
LIN {X 0,Y 597.515,Z 339.219,A -85,B 0,C 180,E1 21634.414,E2 21634.414} C_VEL
LIN {X 0,Y 595.104,Z 334.569,A -85,B 0,C 180,E1 21633.558,E2 21633.558} C_VEL
LIN {X 0,Y 593.391,Z 331.481,A -85,B 0,C 180,E1 21632.951,E2 21632.951} C_VEL
LIN {X 0,Y 593.171,Z 330.479,A -85,B 0,C 180,E1 21632.74,E2 21632.74} C_VEL
LIN {X 0,Y 593.194,Z 330.297,A -85,B 0,C 180,E1 21629.596,E2 21629.596} C_VEL
LIN {X 0,Y 593.163,Z 330.345,A -85,B 0,C 180,E1 21626.425,E2 21626.425} C_VEL
LIN {X 0,Y 593.192,Z 330.296,A -85,B 0,C 180,E1 21623.126,E2 21623.126} C_VEL
LIN {X 0,Y 593.19,Z 330.311,A -85,B 0,C 180,E1 21619.855,E2 21619.855} C_VEL
LIN {X 0,Y 593.174,Z 330.328,A -85,B 0,C 180,E1 21616.552,E2 21616.552} C_VEL
LIN {X 0,Y 593.182,Z 330.294,A -85,B 0,C 180,E1 21613.445,E2 21613.445} C_VEL
LIN {X 0,Y 593.178,Z 330.333,A -85,B 0,C 180,E1 21610.195,E2 21610.195} C_VEL
LIN {X 0,Y 593.179,Z 330.285,A -85,B 0,C 180,E1 21606.971,E2 21606.971} C_VEL
LIN {X 0,Y 593.192,Z 330.337,A -85,B 0,C 180,E1 21603.673,E2 21603.673} C_VEL
LIN {X 0,Y 593.19,Z 330.283,A -85,B 0,C 180,E1 21600.386,E2 21600.386} C_VEL
LIN {X 0,Y 593.172,Z 330.343,A -85,B 0,C 180,E1 21597.101,E2 21597.101} C_VEL
LIN {X 0,Y 593.187,Z 330.285,A -85,B 0,C 180,E1 21593.904,E2 21593.904} C_VEL
LIN {X 0,Y 593.163,Z 330.341,A -85,B 0,C 180,E1 21590.785,E2 21590.785} C_VEL
LIN {X 0,Y 593.189,Z 330.287,A -85,B 0,C 180,E1 21587.54,E2 21587.54} C_VEL
LIN {X 0,Y 593.169,Z 330.341,A -85,B 0,C 180,E1 21584.353,E2 21584.353} C_VEL
LIN {X 0,Y 593.154,Z 330.304,A -85,B 0,C 180,E1 21581.014,E2 21581.014} C_VEL
LIN {X 0,Y 593.189,Z 330.307,A -85,B 0,C 180,E1 21577.92,E2 21577.92} C_VEL
LIN {X 0,Y 593.144,Z 330.337,A -85,B 0,C 180,E1 21574.755,E2 21574.755} C_VEL
LIN {X 0,Y 593.202,Z 330.29,A -85,B 0,C 180,E1 21571.619,E2 21571.619} C_VEL
LIN {X 0,Y 593.169,Z 330.532,A -85,B 0,C 180,E1 21568.792,E2 21568.792} C_VEL
LIN {X 0,Y 594.663,Z 334.104,A -85,B 0,C 180,E1 21568.131,E2 21568.131} C_VEL
LIN {X 0,Y 596.022,Z 336.056,A -85,B 0,C 180,E1 21567.725,E2 21567.725} C_VEL
LIN {X 0,Y 598.269,Z 340.096,A -85,B 0,C 180,E1 21566.986,E2 21566.986} C_VEL
LIN {X 0,Y 600.572,Z 344.568,A -85,B 0,C 180,E1 21566.215,E2 21566.215} C_VEL
LIN {X 0,Y 606.35,Z 355.476,A -85,B 0,C 180,E1 21564.43,E2 21564.43} C_VEL
LIN {X 0,Y 620.495,Z 374.598,A -85,B 0,C 180,E1 21562.415,E2 21562.415} C_VEL
LIN {X 0,Y 631.612,Z 390.391,A -85,B 0,C 180,E1 21560.945,E2 21560.945} C_VEL
LIN {X 0,Y 639.054,Z 401.232,A -85,B 0,C 180,E1 21560.012,E2 21560.012} C_VEL
LIN {X 0,Y 634.209,Z 605.483,A -85,B 0,C 180,E1 21557.162,E2 21557.162} C_VEL
LIN {X 0,Y 629.542,Z 825.704,A -85,B 0,C 180,E1 21554.192,E2 21554.192} C_VEL
LIN {X 0,Y 628.513,Z 848.606,A -85,B 0,C 180,E1 21553.798,E2 21553.798} C_VEL
LIN {X 0,Y 626.923,Z 875.157,A -85,B 0,C 180,E1 21553.187,E2 21553.187} C_VEL
LIN {X 0,Y 624.805,Z 900.4,A -85,B 0,C 180,E1 21552.417,E2 21552.417} C_VEL
LIN {X 0,Y 622.842,Z 921.281,A -85,B 0,C 180,E1 21551.652,E2 21551.652} C_VEL
LIN {X 0,Y 620.752,Z 941.451,A -85,B 0,C 180,E1 21550.794,E2 21550.794} C_VEL
LIN {X 0,Y 618.547,Z 961.065,A -85,B 0,C 180,E1 21549.839,E2 21549.839} C_VEL
LIN {X 0,Y 615.794,Z 983.922,A -85,B 0,C 180,E1 21548.572,E2 21548.572} C_VEL
LIN {X 0,Y 612.643,Z 1007.845,A -85,B 0,C 180,E1 21547.03,E2 21547.03} C_VEL
LIN {X 0,Y 610.048,Z 1027.179,A -85,B 0,C 180,E1 21545.613,E2 21545.613} C_VEL
LIN {X 0,Y 607.525,Z 1045.869,A -85,B 0,C 180,E1 21544.083,E2 21544.083} C_VEL
LIN {X 0,Y 604.605,Z 1067.722,A -85,B 0,C 180,E1 21542.063,E2 21542.063} C_VEL
LIN {X 0,Y 602.202,Z 1085.447,A -85,B 0,C 180,E1 21540.204,E2 21540.204} C_VEL
LIN {X 0,Y 600.131,Z 1101.37,A -85,B 0,C 180,E1 21538.349,E2 21538.349} C_VEL
LIN {X 0,Y 598.08,Z 1118.735,A -85,B 0,C 180,E1 21536.084,E2 21536.084} C_VEL
LIN {X 0,Y 596.283,Z 1134.577,A -85,B 0,C 180,E1 21533.712,E2 21533.712} C_VEL
LIN {X 0,Y 595.034,Z 1147.148,A -85,B 0,C 180,E1 21531.592,E2 21531.592} C_VEL
LIN {X 0,Y 593.898,Z 1160.362,A -85,B 0,C 180,E1 21529.063,E2 21529.063} C_VEL
LIN {X 0,Y 593.098,Z 1171.085,A -85,B 0,C 180,E1 21526.654,E2 21526.654} C_VEL
LIN {X 0,Y 592.634,Z 1179.16,A -85,B 0,C 180,E1 21524.56,E2 21524.56} C_VEL
LIN {X 0,Y 592.284,Z 1186.392,A -85,B 0,C 180,E1 21522.38,E2 21522.38} C_VEL
LIN {X 0,Y 592.069,Z 1193.352,A -85,B 0,C 180,E1 21519.821,E2 21519.821} C_VEL
LIN {X 0,Y 591.963,Z 1198.748,A -85,B 0,C 180,E1 21517.18,E2 21517.18} C_VEL
LIN {X 0,Y 591.92,Z 1202.115,A -85,B 0,C 180,E1 21514.845,E2 21514.845} C_VEL
LIN {X 0,Y 591.908,Z 1204.197,A -85,B 0,C 180,E1 21512.517,E2 21512.517} C_VEL
LIN {X 0,Y 591.901,Z 1204.961,A -85,B 0,C 180,E1 21509.806,E2 21509.806} C_VEL
LIN {X 0,Y 591.912,Z 1204.06,A -85,B 0,C 180,E1 21507.289,E2 21507.289} C_VEL
LIN {X 0,Y 591.925,Z 1201.887,A -85,B 0,C 180,E1 21504.961,E2 21504.961} C_VEL
LIN {X 0,Y 591.968,Z 1198.078,A -85,B 0,C 180,E1 21502.429,E2 21502.429} C_VEL
LIN {X 0,Y 592.095,Z 1192.368,A -85,B 0,C 180,E1 21499.786,E2 21499.786} C_VEL
LIN {X 0,Y 592.315,Z 1185.783,A -85,B 0,C 180,E1 21497.422,E2 21497.422} C_VEL
LIN {X 0,Y 592.695,Z 1178.09,A -85,B 0,C 180,E1 21495.142,E2 21495.142} C_VEL
LIN {X 0,Y 593.373,Z 1167.283,A -85,B 0,C 180,E1 21492.444,E2 21492.444} C_VEL
LIN {X 0,Y 594.221,Z 1156.301,A -85,B 0,C 180,E1 21490.129,E2 21490.129} C_VEL
LIN {X 0,Y 595.249,Z 1144.856,A -85,B 0,C 180,E1 21488.001,E2 21488.001} C_VEL
LIN {X 0,Y 596.804,Z 1129.967,A -85,B 0,C 180,E1 21485.555,E2 21485.555} C_VEL
LIN {X 0,Y 598.576,Z 1114.151,A -85,B 0,C 180,E1 21483.298,E2 21483.298} C_VEL
LIN {X 0,Y 600.453,Z 1098.907,A -85,B 0,C 180,E1 21481.352,E2 21481.352} C_VEL
LIN {X 0,Y 602.856,Z 1080.8,A -85,B 0,C 180,E1 21479.28,E2 21479.28} C_VEL
LIN {X 0,Y 605.506,Z 1060.709,A -85,B 0,C 180,E1 21477.261,E2 21477.261} C_VEL
LIN {X 0,Y 607.839,Z 1043.427,A -85,B 0,C 180,E1 21475.708,E2 21475.708} C_VEL
LIN {X 0,Y 610.367,Z 1024.875,A -85,B 0,C 180,E1 21474.209,E2 21474.209} C_VEL
LIN {X 0,Y 613.561,Z 1001.363,A -85,B 0,C 180,E1 21472.527,E2 21472.527} C_VEL
LIN {X 0,Y 616.4,Z 978.838,A -85,B 0,C 180,E1 21471.136,E2 21471.136} C_VEL
LIN {X 0,Y 618.709,Z 959.678,A -85,B 0,C 180,E1 21470.09,E2 21470.09} C_VEL
LIN {X 0,Y 620.853,Z 940.57,A -85,B 0,C 180,E1 21469.167,E2 21469.167} C_VEL
LIN {X 0,Y 622.974,Z 919.984,A -85,B 0,C 180,E1 21468.296,E2 21468.296} C_VEL
LIN {X 0,Y 625.163,Z 896.691,A -85,B 0,C 180,E1 21467.457,E2 21467.457} C_VEL
LIN {X 0,Y 627.305,Z 869.096,A -85,B 0,C 180,E1 21466.659,E2 21466.659} C_VEL
LIN {X 0,Y 628.609,Z 846.555,A -85,B 0,C 180,E1 21466.162,E2 21466.162} C_VEL
LIN {X 0,Y 629.582,Z 824.494,A -85,B 0,C 180,E1 21465.79,E2 21465.79} C_VEL
LIN {X 0,Y 634.248,Z 603.573,A -85,B 0,C 180,E1 21462.812,E2 21462.812} C_VEL
LIN {X 0,Y 638.903,Z 407.246,A -85,B 0,C 180,E1 21460.073,E2 21460.073} C_VEL
LIN {X 0,Y 638.937,Z 400.922,A -85,B 0,C 180,E1 21459.971,E2 21459.971} C_VEL
LIN {X 0,Y 622.467,Z 377.292,A -85,B 0,C 180,E1 21457.852,E2 21457.852} C_VEL
LIN {X 0,Y 608.432,Z 358.29,A -85,B 0,C 180,E1 21455.891,E2 21455.891} C_VEL
LIN {X 0,Y 606.039,Z 354.92,A -85,B 0,C 180,E1 21455.504,E2 21455.504} C_VEL
LIN {X 0,Y 600.207,Z 344.084,A -85,B 0,C 180,E1 21453.694,E2 21453.694} C_VEL
LIN {X 0,Y 597.565,Z 339.196,A -85,B 0,C 180,E1 21452.83,E2 21452.83} C_VEL
LIN {X 0,Y 595.312,Z 334.886,A -85,B 0,C 180,E1 21452.057,E2 21452.057} C_VEL
LIN {X 0,Y 593.522,Z 331.993,A -85,B 0,C 180,E1 21451.483,E2 21451.483} C_VEL
LIN {X 0,Y 593.161,Z 330.476,A -85,B 0,C 180,E1 21451.166,E2 21451.166} C_VEL
LIN {X 0,Y 593.143,Z 330.299,A -85,B 0,C 180,E1 21447.837,E2 21447.837} C_VEL
LIN {X 0,Y 593.17,Z 330.318,A -85,B 0,C 180,E1 21444.818,E2 21444.818} C_VEL
LIN {X 0,Y 593.147,Z 330.328,A -85,B 0,C 180,E1 21441.561,E2 21441.561} C_VEL
LIN {X 0,Y 593.19,Z 330.291,A -85,B 0,C 180,E1 21438.475,E2 21438.475} C_VEL
LIN {X 0,Y 593.152,Z 330.344,A -85,B 0,C 180,E1 21435.247,E2 21435.247} C_VEL
LIN {X 0,Y 593.192,Z 330.286,A -85,B 0,C 180,E1 21432.065,E2 21432.065} C_VEL
LIN {X 0,Y 593.167,Z 330.344,A -85,B 0,C 180,E1 21428.824,E2 21428.824} C_VEL
LIN {X 0,Y 593.18,Z 330.29,A -85,B 0,C 180,E1 21425.514,E2 21425.514} C_VEL
LIN {X 0,Y 593.191,Z 330.334,A -85,B 0,C 180,E1 21422.319,E2 21422.319} C_VEL
LIN {X 0,Y 593.168,Z 330.292,A -85,B 0,C 180,E1 21419.034,E2 21419.034} C_VEL
LIN {X 0,Y 593.186,Z 330.33,A -85,B 0,C 180,E1 21415.843,E2 21415.843} C_VEL
LIN {X 0,Y 593.174,Z 330.29,A -85,B 0,C 180,E1 21412.64,E2 21412.64} C_VEL
LIN {X 0,Y 593.187,Z 330.327,A -85,B 0,C 180,E1 21409.413,E2 21409.413} C_VEL
LIN {X 0,Y 593.189,Z 330.303,A -85,B 0,C 180,E1 21406.052,E2 21406.052} C_VEL
LIN {X 0,Y 593.189,Z 330.306,A -85,B 0,C 180,E1 21402.843,E2 21402.843} C_VEL
LIN {X 0,Y 593.171,Z 330.33,A -85,B 0,C 180,E1 21399.578,E2 21399.578} C_VEL
LIN {X 0,Y 593.188,Z 330.292,A -85,B 0,C 180,E1 21396.453,E2 21396.453} C_VEL
LIN {X 0,Y 593.167,Z 330.343,A -85,B 0,C 180,E1 21393.251,E2 21393.251} C_VEL
LIN {X 0,Y 593.197,Z 330.302,A -85,B 0,C 180,E1 21390.041,E2 21390.041} C_VEL
LIN {X 0,Y 593.185,Z 330.521,A -85,B 0,C 180,E1 21387.127,E2 21387.127} C_VEL
LIN {X 0,Y 594.805,Z 334.202,A -85,B 0,C 180,E1 21386.422,E2 21386.422} C_VEL
LIN {X 0,Y 595.98,Z 336.161,A -85,B 0,C 180,E1 21386.035,E2 21386.035} C_VEL
LIN {X 0,Y 599.026,Z 342.183,A -85,B 0,C 180,E1 21384.956,E2 21384.956} C_VEL
LIN {X 0,Y 601.136,Z 346.056,A -85,B 0,C 180,E1 21384.262,E2 21384.262} C_VEL
LIN {X 0,Y 607.39,Z 358.172,A -85,B 0,C 180,E1 21382.237,E2 21382.237} C_VEL
LIN {X 0,Y 615.453,Z 374.902,A -85,B 0,C 180,E1 21379.713,E2 21379.713} C_VEL
LIN {X 0,Y 623.323,Z 392.387,A -85,B 0,C 180,E1 21377.363,E2 21377.363} C_VEL
LIN {X 0,Y 625.784,Z 396.725,A -85,B 0,C 180,E1 21377.022,E2 21377.022} C_VEL
LIN {X 0,Y 633.945,Z 436.394,A -85,B 0,C 180,E1 21375.531,E2 21375.531} C_VEL
LIN {X 0,Y 631.458,Z 541.457,A -85,B 0,C 180,E1 21374.107,E2 21374.107} C_VEL
LIN {X 0,Y 630.607,Z 549.162,A -85,B 0,C 180,E1 21374.068,E2 21374.068} C_VEL
LIN {X 0,Y 625.808,Z 569.811,A -85,B 0,C 180,E1 21374.205,E2 21374.205} C_VEL
LIN {X 0,Y 625.134,Z 576.423,A -85,B 0,C 180,E1 21374.165,E2 21374.165} C_VEL
LIN {X 0,Y 619.904,Z 803.456,A -85,B 0,C 180,E1 21371.121,E2 21371.121} C_VEL
LIN {X 0,Y 618.764,Z 839.19,A -85,B 0,C 180,E1 21370.598,E2 21370.598} C_VEL
LIN {X 0,Y 617.359,Z 861.919,A -85,B 0,C 180,E1 21370.125,E2 21370.125} C_VEL
LIN {X 0,Y 615.81,Z 882.332,A -85,B 0,C 180,E1 21369.579,E2 21369.579} C_VEL
LIN {X 0,Y 613.925,Z 903.336,A -85,B 0,C 180,E1 21368.892,E2 21368.892} C_VEL
LIN {X 0,Y 611.338,Z 928.323,A -85,B 0,C 180,E1 21367.89,E2 21367.89} C_VEL
LIN {X 0,Y 608.864,Z 949.125,A -85,B 0,C 180,E1 21366.892,E2 21366.892} C_VEL
LIN {X 0,Y 606.526,Z 967.526,A -85,B 0,C 180,E1 21365.878,E2 21365.878} C_VEL
LIN {X 0,Y 603.737,Z 988.505,A -85,B 0,C 180,E1 21364.558,E2 21364.558} C_VEL
LIN {X 0,Y 600.635,Z 1010.358,A -85,B 0,C 180,E1 21362.963,E2 21362.963} C_VEL
LIN {X 0,Y 598.126,Z 1027.923,A -85,B 0,C 180,E1 21361.507,E2 21361.507} C_VEL
LIN {X 0,Y 595.118,Z 1050.089,A -85,B 0,C 180,E1 21359.435,E2 21359.435} C_VEL
LIN {X 0,Y 593.008,Z 1066.384,A -85,B 0,C 180,E1 21357.721,E2 21357.721} C_VEL
LIN {X 0,Y 591.072,Z 1082.077,A -85,B 0,C 180,E1 21355.877,E2 21355.877} C_VEL
LIN {X 0,Y 589.061,Z 1099.33,A -85,B 0,C 180,E1 21353.564,E2 21353.564} C_VEL
LIN {X 0,Y 587.658,Z 1112.411,A -85,B 0,C 180,E1 21351.563,E2 21351.563} C_VEL
LIN {X 0,Y 586.389,Z 1125.953,A -85,B 0,C 180,E1 21349.214,E2 21349.214} C_VEL
LIN {X 0,Y 585.472,Z 1136.941,A -85,B 0,C 180,E1 21346.98,E2 21346.98} C_VEL
LIN {X 0,Y 584.9,Z 1145.602,A -85,B 0,C 180,E1 21344.959,E2 21344.959} C_VEL
LIN {X 0,Y 584.416,Z 1154.47,A -85,B 0,C 180,E1 21342.55,E2 21342.55} C_VEL
LIN {X 0,Y 584.12,Z 1161.516,A -85,B 0,C 180,E1 21340.155,E2 21340.155} C_VEL
LIN {X 0,Y 584.007,Z 1166.44,A -85,B 0,C 180,E1 21338.071,E2 21338.071} C_VEL
LIN {X 0,Y 583.929,Z 1170.235,A -85,B 0,C 180,E1 21335.996,E2 21335.996} C_VEL
LIN {X 0,Y 583.901,Z 1173.357,A -85,B 0,C 180,E1 21333.535,E2 21333.535} C_VEL
LIN {X 0,Y 583.911,Z 1174.745,A -85,B 0,C 180,E1 21331.08,E2 21331.08} C_VEL
LIN {X 0,Y 583.908,Z 1174.79,A -85,B 0,C 180,E1 21329.019,E2 21329.019} C_VEL
LIN {X 0,Y 583.906,Z 1173.766,A -85,B 0,C 180,E1 21326.957,E2 21326.957} C_VEL
LIN {X 0,Y 583.919,Z 1171.015,A -85,B 0,C 180,E1 21324.399,E2 21324.399} C_VEL
LIN {X 0,Y 584.002,Z 1166.835,A -85,B 0,C 180,E1 21322.029,E2 21322.029} C_VEL
LIN {X 0,Y 584.101,Z 1162.001,A -85,B 0,C 180,E1 21319.945,E2 21319.945} C_VEL
LIN {X 0,Y 584.376,Z 1155.388,A -85,B 0,C 180,E1 21317.651,E2 21317.651} C_VEL
LIN {X 0,Y 584.852,Z 1146.372,A -85,B 0,C 180,E1 21315.141,E2 21315.141} C_VEL
LIN {X 0,Y 585.437,Z 1137.388,A -85,B 0,C 180,E1 21313.028,E2 21313.028} C_VEL
LIN {X 0,Y 586.344,Z 1126.408,A -85,B 0,C 180,E1 21310.785,E2 21310.785} C_VEL
LIN {X 0,Y 587.605,Z 1112.961,A -85,B 0,C 180,E1 21308.436,E2 21308.436} C_VEL
LIN {X 0,Y 588.942,Z 1100.288,A -85,B 0,C 180,E1 21306.486,E2 21306.486} C_VEL
LIN {X 0,Y 590.817,Z 1084.483,A -85,B 0,C 180,E1 21304.327,E2 21304.327} C_VEL
LIN {X 0,Y 592.878,Z 1067.41,A -85,B 0,C 180,E1 21302.303,E2 21302.303} C_VEL
LIN {X 0,Y 594.879,Z 1051.826,A -85,B 0,C 180,E1 21300.651,E2 21300.651} C_VEL
LIN {X 0,Y 597.939,Z 1029.288,A -85,B 0,C 180,E1 21298.522,E2 21298.522} C_VEL
LIN {X 0,Y 600.396,Z 1011.947,A -85,B 0,C 180,E1 21297.072,E2 21297.072} C_VEL
LIN {X 0,Y 603.367,Z 991.194,A -85,B 0,C 180,E1 21295.534,E2 21295.534} C_VEL
LIN {X 0,Y 606.359,Z 968.872,A -85,B 0,C 180,E1 21294.111,E2 21294.111} C_VEL
LIN {X 0,Y 608.658,Z 950.81,A -85,B 0,C 180,E1 21293.106,E2 21293.106} C_VEL
LIN {X 0,Y 610.88,Z 932.165,A -85,B 0,C 180,E1 21292.195,E2 21292.195} C_VEL
LIN {X 0,Y 613.376,Z 909.586,A -85,B 0,C 180,E1 21291.247,E2 21291.247} C_VEL
LIN {X 0,Y 615.637,Z 884.668,A -85,B 0,C 180,E1 21290.4,E2 21290.4} C_VEL
LIN {X 0,Y 617.224,Z 864.095,A -85,B 0,C 180,E1 21289.839,E2 21289.839} C_VEL
LIN {X 0,Y 618.459,Z 844.384,A -85,B 0,C 180,E1 21289.411,E2 21289.411} C_VEL
LIN {X 0,Y 619.562,Z 818.298,A -85,B 0,C 180,E1 21288.987,E2 21288.987} C_VEL
LIN {X 0,Y 624.875,Z 588.205,A -85,B 0,C 180,E1 21285.904,E2 21285.904} C_VEL
LIN {X 0,Y 628.438,Z 437.645,A -85,B 0,C 180,E1 21283.842,E2 21283.842} C_VEL
LIN {X 0,Y 620.852,Z 400.813,A -85,B 0,C 180,E1 21282.424,E2 21282.424} C_VEL
LIN {X 0,Y 614.596,Z 390.992,A -85,B 0,C 180,E1 21281.527,E2 21281.527} C_VEL
LIN {X 0,Y 607.183,Z 374.832,A -85,B 0,C 180,E1 21279.225,E2 21279.225} C_VEL
LIN {X 0,Y 599.658,Z 359.192,A -85,B 0,C 180,E1 21276.771,E2 21276.771} C_VEL
LIN {X 0,Y 594.328,Z 349.123,A -85,B 0,C 180,E1 21275.008,E2 21275.008} C_VEL
LIN {X 0,Y 592.056,Z 344.812,A -85,B 0,C 180,E1 21274.221,E2 21274.221} C_VEL
LIN {X 0,Y 589.89,Z 340.512,A -85,B 0,C 180,E1 21273.428,E2 21273.428} C_VEL
LIN {X 0,Y 587.985,Z 336.946,A -85,B 0,C 180,E1 21272.736,E2 21272.736} C_VEL
LIN {X 0,Y 585.539,Z 332.636,A -85,B 0,C 180,E1 21271.848,E2 21271.848} C_VEL
LIN {X 0,Y 585.283,Z 331.472,A -85,B 0,C 180,E1 21271.576,E2 21271.576} C_VEL
LIN {X 0,Y 585.217,Z 331.283,A -85,B 0,C 180,E1 21268.47,E2 21268.47} C_VEL
LIN {X 0,Y 585.25,Z 331.297,A -85,B 0,C 180,E1 21265.177,E2 21265.177} C_VEL
LIN {X 0,Y 585.258,Z 331.317,A -85,B 0,C 180,E1 21261.867,E2 21261.867} C_VEL
LIN {X 0,Y 585.228,Z 331.277,A -85,B 0,C 180,E1 21258.529,E2 21258.529} C_VEL
LIN {X 0,Y 585.25,Z 331.329,A -85,B 0,C 180,E1 21255.356,E2 21255.356} C_VEL
LIN {X 0,Y 585.234,Z 331.273,A -85,B 0,C 180,E1 21252.131,E2 21252.131} C_VEL
LIN {X 0,Y 585.255,Z 331.322,A -85,B 0,C 180,E1 21248.845,E2 21248.845} C_VEL
LIN {X 0,Y 585.241,Z 331.278,A -85,B 0,C 180,E1 21245.49,E2 21245.49} C_VEL
LIN {X 0,Y 585.248,Z 331.312,A -85,B 0,C 180,E1 21242.252,E2 21242.252} C_VEL
LIN {X 0,Y 585.23,Z 331.286,A -85,B 0,C 180,E1 21239.021,E2 21239.021} C_VEL
LIN {X 0,Y 585.251,Z 331.307,A -85,B 0,C 180,E1 21235.787,E2 21235.787} C_VEL
LIN {X 0,Y 585.237,Z 331.292,A -85,B 0,C 180,E1 21232.539,E2 21232.539} C_VEL
LIN {X 0,Y 585.227,Z 331.295,A -85,B 0,C 180,E1 21229.167,E2 21229.167} C_VEL
LIN {X 0,Y 585.259,Z 331.309,A -85,B 0,C 180,E1 21225.96,E2 21225.96} C_VEL
LIN {X 0,Y 585.209,Z 331.285,A -85,B 0,C 180,E1 21222.764,E2 21222.764} C_VEL
LIN {X 0,Y 585.26,Z 331.329,A -85,B 0,C 180,E1 21219.498,E2 21219.498} C_VEL
LIN {X 0,Y 585.2,Z 331.283,A -85,B 0,C 180,E1 21216.433,E2 21216.433} C_VEL
LIN {X 0,Y 585.236,Z 331.302,A -85,B 0,C 180,E1 21213.189,E2 21213.189} C_VEL
LIN {X 0,Y 585.207,Z 331.367,A -85,B 0,C 180,E1 21210.185,E2 21210.185} C_VEL
LIN {X 0,Y 585.324,Z 331.906,A -85,B 0,C 180,E1 21209.852,E2 21209.852} C_VEL
LIN {X 0,Y 587.187,Z 335.638,A -85,B 0,C 180,E1 21209.117,E2 21209.117} C_VEL
LIN {X 0,Y 588.187,Z 337.424,A -85,B 0,C 180,E1 21208.766,E2 21208.766} C_VEL
LIN {X 0,Y 590.277,Z 340.995,A -85,B 0,C 180,E1 21208.065,E2 21208.065} C_VEL
LIN {X 0,Y 593.908,Z 348.1,A -85,B 0,C 180,E1 21206.796,E2 21206.796} C_VEL
LIN {X 0,Y 598.159,Z 355.812,A -85,B 0,C 180,E1 21205.452,E2 21205.452} C_VEL
LIN {X 0,Y 613.092,Z 375.661,A -85,B 0,C 180,E1 21203.234,E2 21203.234} C_VEL
LIN {X 0,Y 626.718,Z 395.084,A -85,B 0,C 180,E1 21201.375,E2 21201.375} C_VEL
LIN {X 0,Y 633.557,Z 405.194,A -85,B 0,C 180,E1 21200.492,E2 21200.492} C_VEL
LIN {X 0,Y 628.394,Z 608.97,A -85,B 0,C 180,E1 21197.624,E2 21197.624} C_VEL
LIN {X 0,Y 623.396,Z 827.266,A -85,B 0,C 180,E1 21194.647,E2 21194.647} C_VEL
LIN {X 0,Y 622.088,Z 854.38,A -85,B 0,C 180,E1 21194.161,E2 21194.161} C_VEL
LIN {X 0,Y 620.217,Z 881.339,A -85,B 0,C 180,E1 21193.489,E2 21193.489} C_VEL
LIN {X 0,Y 618.486,Z 902.819,A -85,B 0,C 180,E1 21192.828,E2 21192.828} C_VEL
LIN {X 0,Y 616.844,Z 920.621,A -85,B 0,C 180,E1 21192.182,E2 21192.182} C_VEL
LIN {X 0,Y 614.685,Z 940.572,A -85,B 0,C 180,E1 21191.332,E2 21191.332} C_VEL
LIN {X 0,Y 612.543,Z 958.672,A -85,B 0,C 180,E1 21190.455,E2 21190.455} C_VEL
LIN {X 0,Y 610.139,Z 977.624,A -85,B 0,C 180,E1 21189.421,E2 21189.421} C_VEL
LIN {X 0,Y 607.446,Z 997.859,A -85,B 0,C 180,E1 21188.176,E2 21188.176} C_VEL
LIN {X 0,Y 603.997,Z 1022.554,A -85,B 0,C 180,E1 21186.433,E2 21186.433} C_VEL
LIN {X 0,Y 601.133,Z 1042.218,A -85,B 0,C 180,E1 21184.844,E2 21184.844} C_VEL
LIN {X 0,Y 598.621,Z 1059.602,A -85,B 0,C 180,E1 21183.277,E2 21183.277} C_VEL
LIN {X 0,Y 595.845,Z 1079.328,A -85,B 0,C 180,E1 21181.295,E2 21181.295} C_VEL
LIN {X 0,Y 593.242,Z 1097.987,A -85,B 0,C 180,E1 21179.149,E2 21179.149} C_VEL
LIN {X 0,Y 591.278,Z 1112.612,A -85,B 0,C 180,E1 21177.275,E2 21177.275} C_VEL
LIN {X 0,Y 589.498,Z 1127.184,A -85,B 0,C 180,E1 21175.197,E2 21175.197} C_VEL
LIN {X 0,Y 587.643,Z 1143.704,A -85,B 0,C 180,E1 21172.509,E2 21172.509} C_VEL
LIN {X 0,Y 586.477,Z 1155.376,A -85,B 0,C 180,E1 21170.33,E2 21170.33} C_VEL
LIN {X 0,Y 585.631,Z 1165.447,A -85,B 0,C 180,E1 21168.206,E2 21168.206} C_VEL
LIN {X 0,Y 584.858,Z 1176.307,A -85,B 0,C 180,E1 21165.569,E2 21165.569} C_VEL
LIN {X 0,Y 584.39,Z 1185.176,A -85,B 0,C 180,E1 21162.952,E2 21162.952} C_VEL
LIN {X 0,Y 584.128,Z 1191.603,A -85,B 0,C 180,E1 21160.653,E2 21160.653} C_VEL
LIN {X 0,Y 583.992,Z 1197.151,A -85,B 0,C 180,E1 21158.17,E2 21158.17} C_VEL
LIN {X 0,Y 583.93,Z 1201.428,A -85,B 0,C 180,E1 21155.502,E2 21155.502} C_VEL
LIN {X 0,Y 583.917,Z 1203.854,A -85,B 0,C 180,E1 21153.043,E2 21153.043} C_VEL
LIN {X 0,Y 583.905,Z 1204.804,A -85,B 0,C 180,E1 21150.883,E2 21150.883} C_VEL
LIN {X 0,Y 583.915,Z 1204.736,A -85,B 0,C 180,E1 21148.822,E2 21148.822} C_VEL
LIN {X 0,Y 583.913,Z 1203.51,A -85,B 0,C 180,E1 21146.466,E2 21146.466} C_VEL
LIN {X 0,Y 583.944,Z 1200.336,A -85,B 0,C 180,E1 21143.708,E2 21143.708} C_VEL
LIN {X 0,Y 584.018,Z 1195.925,A -85,B 0,C 180,E1 21141.235,E2 21141.235} C_VEL
LIN {X 0,Y 584.152,Z 1190.584,A -85,B 0,C 180,E1 21138.947,E2 21138.947} C_VEL
LIN {X 0,Y 584.519,Z 1182.683,A -85,B 0,C 180,E1 21136.245,E2 21136.245} C_VEL
LIN {X 0,Y 585.07,Z 1173.111,A -85,B 0,C 180,E1 21133.621,E2 21133.621} C_VEL
LIN {X 0,Y 585.743,Z 1164.072,A -85,B 0,C 180,E1 21131.488,E2 21131.488} C_VEL
LIN {X 0,Y 586.694,Z 1153.203,A -85,B 0,C 180,E1 21129.238,E2 21129.238} C_VEL
LIN {X 0,Y 588.228,Z 1138.273,A -85,B 0,C 180,E1 21126.562,E2 21126.562} C_VEL
LIN {X 0,Y 589.784,Z 1124.558,A -85,B 0,C 180,E1 21124.413,E2 21124.413} C_VEL
LIN {X 0,Y 591.602,Z 1110.296,A -85,B 0,C 180,E1 21122.413,E2 21122.413} C_VEL
LIN {X 0,Y 594.106,Z 1091.615,A -85,B 0,C 180,E1 21120.084,E2 21120.084} C_VEL
LIN {X 0,Y 596.593,Z 1073.801,A -85,B 0,C 180,E1 21118.134,E2 21118.134} C_VEL
LIN {X 0,Y 598.95,Z 1057.377,A -85,B 0,C 180,E1 21116.514,E2 21116.514} C_VEL
LIN {X 0,Y 601.696,Z 1038.575,A -85,B 0,C 180,E1 21114.846,E2 21114.846} C_VEL
LIN {X 0,Y 605.031,Z 1015.173,A -85,B 0,C 180,E1 21113.019,E2 21113.019} C_VEL
LIN {X 0,Y 607.752,Z 995.41,A -85,B 0,C 180,E1 21111.666,E2 21111.666} C_VEL
LIN {X 0,Y 610.363,Z 975.817,A -85,B 0,C 180,E1 21110.474,E2 21110.474} C_VEL
LIN {X 0,Y 612.908,Z 955.655,A -85,B 0,C 180,E1 21109.389,E2 21109.389} C_VEL
LIN {X 0,Y 615.759,Z 931.513,A -85,B 0,C 180,E1 21108.259,E2 21108.259} C_VEL
LIN {X 0,Y 618.107,Z 907.427,A -85,B 0,C 180,E1 21107.328,E2 21107.328} C_VEL
LIN {X 0,Y 619.93,Z 885.188,A -85,B 0,C 180,E1 21106.621,E2 21106.621} C_VEL
LIN {X 0,Y 621.448,Z 863.781,A -85,B 0,C 180,E1 21106.059,E2 21106.059} C_VEL
LIN {X 0,Y 622.705,Z 842.065,A -85,B 0,C 180,E1 21105.601,E2 21105.601} C_VEL
LIN {X 0,Y 623.855,Z 814.269,A -85,B 0,C 180,E1 21105.162,E2 21105.162} C_VEL
LIN {X 0,Y 628.652,Z 597.148,A -85,B 0,C 180,E1 21102.215,E2 21102.215} C_VEL
LIN {X 0,Y 633.557,Z 404.931,A -85,B 0,C 180,E1 21099.503,E2 21099.503} C_VEL
LIN {X 0,Y 618.218,Z 382.917,A -85,B 0,C 180,E1 21097.484,E2 21097.484} C_VEL
LIN {X 0,Y 605.009,Z 364.847,A -85,B 0,C 180,E1 21095.603,E2 21095.603} C_VEL
LIN {X 0,Y 598.074,Z 355.617,A -85,B 0,C 180,E1 21094.525,E2 21094.525} C_VEL
LIN {X 0,Y 592.398,Z 345.138,A -85,B 0,C 180,E1 21092.692,E2 21092.692} C_VEL
LIN {X 0,Y 590.153,Z 340.858,A -85,B 0,C 180,E1 21091.912,E2 21091.912} C_VEL
LIN {X 0,Y 588.144,Z 337.31,A -85,B 0,C 180,E1 21091.226,E2 21091.226} C_VEL
LIN {X 0,Y 586.699,Z 335.015,A -85,B 0,C 180,E1 21090.749,E2 21090.749} C_VEL
LIN {X 0,Y 585.241,Z 331.496,A -85,B 0,C 180,E1 21090.039,E2 21090.039} C_VEL
LIN {X 0,Y 585.197,Z 331.295,A -85,B 0,C 180,E1 21087.253,E2 21087.253} C_VEL
LIN {X 0,Y 585.239,Z 331.285,A -85,B 0,C 180,E1 21084.1,E2 21084.1} C_VEL
LIN {X 0,Y 585.215,Z 331.331,A -85,B 0,C 180,E1 21081.027,E2 21081.027} C_VEL
LIN {X 0,Y 585.223,Z 331.278,A -85,B 0,C 180,E1 21077.706,E2 21077.706} C_VEL
LIN {X 0,Y 585.252,Z 331.323,A -85,B 0,C 180,E1 21074.545,E2 21074.545} C_VEL
LIN {X 0,Y 585.215,Z 331.286,A -85,B 0,C 180,E1 21071.232,E2 21071.232} C_VEL
LIN {X 0,Y 585.255,Z 331.311,A -85,B 0,C 180,E1 21068.053,E2 21068.053} C_VEL
LIN {X 0,Y 585.225,Z 331.292,A -85,B 0,C 180,E1 21064.802,E2 21064.802} C_VEL
LIN {X 0,Y 585.253,Z 331.303,A -85,B 0,C 180,E1 21061.566,E2 21061.566} C_VEL
LIN {X 0,Y 585.251,Z 331.295,A -85,B 0,C 180,E1 21058.238,E2 21058.238} C_VEL
LIN {X 0,Y 585.235,Z 331.293,A -85,B 0,C 180,E1 21055.001,E2 21055.001} C_VEL
LIN {X 0,Y 585.242,Z 331.297,A -85,B 0,C 180,E1 21051.848,E2 21051.848} C_VEL
LIN {X 0,Y 585.24,Z 331.287,A -85,B 0,C 180,E1 21048.669,E2 21048.669} C_VEL
LIN {X 0,Y 585.241,Z 331.311,A -85,B 0,C 180,E1 21045.454,E2 21045.454} C_VEL
LIN {X 0,Y 585.249,Z 331.278,A -85,B 0,C 180,E1 21042.192,E2 21042.192} C_VEL
LIN {X 0,Y 585.26,Z 331.329,A -85,B 0,C 180,E1 21038.87,E2 21038.87} C_VEL
LIN {X 0,Y 585.225,Z 331.283,A -85,B 0,C 180,E1 21035.577,E2 21035.577} C_VEL
LIN {X 0,Y 585.255,Z 331.296,A -85,B 0,C 180,E1 21032.419,E2 21032.419} C_VEL
LIN {X 0,Y 585.222,Z 331.319,A -85,B 0,C 180,E1 21029.249,E2 21029.249} C_VEL
LIN {X 0,Y 585.315,Z 331.696,A -85,B 0,C 180,E1 21028.213,E2 21028.213} C_VEL
LIN {X 0,Y 586.829,Z 335.195,A -85,B 0,C 180,E1 21027.539,E2 21027.539} C_VEL
LIN {X 0,Y 588.03,Z 337.05,A -85,B 0,C 180,E1 21027.139,E2 21027.139} C_VEL
LIN {X 0,Y 590.258,Z 340.96,A -85,B 0,C 180,E1 21026.362,E2 21026.362} C_VEL
LIN {X 0,Y 592.418,Z 345.318,A -85,B 0,C 180,E1 21025.568,E2 21025.568} C_VEL
LIN {X 0,Y 597.888,Z 355.879,A -85,B 0,C 180,E1 21023.699,E2 21023.699} C_VEL
LIN {X 0,Y 605.742,Z 371.645,A -85,B 0,C 180,E1 21021.151,E2 21021.151} C_VEL
LIN {X 0,Y 613.835,Z 389.413,A -85,B 0,C 180,E1 21018.597,E2 21018.597} C_VEL
LIN {X 0,Y 615.543,Z 392.647,A -85,B 0,C 180,E1 21018.212,E2 21018.212} C_VEL
LIN {X 0,Y 621.044,Z 401.418,A -85,B 0,C 180,E1 21017.452,E2 21017.452} C_VEL
LIN {X 0,Y 628.522,Z 438.426,A -85,B 0,C 180,E1 21016.045,E2 21016.045} C_VEL
LIN {X 0,Y 625.134,Z 576.423,A -85,B 0,C 180,E1 21014.165,E2 21014.165} C_VEL
LIN {X 0,Y 624.268,Z 584.13,A -85,B 0,C 180,E1 21014.127,E2 21014.127} C_VEL
LIN {X 0,Y 619.464,Z 604.776,A -85,B 0,C 180,E1 21014.267,E2 21014.267} C_VEL
LIN {X 0,Y 618.786,Z 611.389,A -85,B 0,C 180,E1 21014.228,E2 21014.228} C_VEL
LIN {X 0,Y 613.535,Z 827.43,A -85,B 0,C 180,E1 21011.314,E2 21011.314} C_VEL
LIN {X 0,Y 612.484,Z 848.975,A -85,B 0,C 180,E1 21010.938,E2 21010.938} C_VEL
LIN {X 0,Y 610.974,Z 871.599,A -85,B 0,C 180,E1 21010.415,E2 21010.415} C_VEL
LIN {X 0,Y 608.724,Z 896.713,A -85,B 0,C 180,E1 21009.654,E2 21009.654} C_VEL
LIN {X 0,Y 606.632,Z 916.86,A -85,B 0,C 180,E1 21008.902,E2 21008.902} C_VEL
LIN {X 0,Y 604.365,Z 936.389,A -85,B 0,C 180,E1 21008.046,E2 21008.046} C_VEL
LIN {X 0,Y 601.46,Z 959.214,A -85,B 0,C 180,E1 21006.88,E2 21006.88} C_VEL
LIN {X 0,Y 598.244,Z 981.701,A -85,B 0,C 180,E1 21005.515,E2 21005.515} C_VEL
LIN {X 0,Y 595.523,Z 1000.28,A -85,B 0,C 180,E1 21004.226,E2 21004.226} C_VEL
LIN {X 0,Y 592.226,Z 1022.363,A -85,B 0,C 180,E1 21002.472,E2 21002.472} C_VEL
LIN {X 0,Y 589.56,Z 1039.825,A -85,B 0,C 180,E1 21000.887,E2 21000.887} C_VEL
LIN {X 0,Y 587.141,Z 1055.882,A -85,B 0,C 180,E1 20999.259,E2 20999.259} C_VEL
LIN {X 0,Y 584.25,Z 1077.01,A -85,B 0,C 180,E1 20996.86,E2 20996.86} C_VEL
LIN {X 0,Y 582.478,Z 1090.807,A -85,B 0,C 180,E1 20995.087,E2 20995.087} C_VEL
LIN {X 0,Y 580.766,Z 1105.299,A -85,B 0,C 180,E1 20993.005,E2 20993.005} C_VEL
LIN {X 0,Y 579.184,Z 1119.694,A -85,B 0,C 180,E1 20990.621,E2 20990.621} C_VEL
LIN {X 0,Y 578.144,Z 1130.601,A -85,B 0,C 180,E1 20988.556,E2 20988.556} C_VEL
LIN {X 0,Y 577.277,Z 1141.526,A -85,B 0,C 180,E1 20986.192,E2 20986.192} C_VEL
LIN {X 0,Y 576.64,Z 1150.939,A -85,B 0,C 180,E1 20983.742,E2 20983.742} C_VEL
LIN {X 0,Y 576.292,Z 1157.85,A -85,B 0,C 180,E1 20981.611,E2 20981.611} C_VEL
LIN {X 0,Y 576.074,Z 1164.317,A -85,B 0,C 180,E1 20979.189,E2 20979.189} C_VEL
LIN {X 0,Y 575.946,Z 1169.274,A -85,B 0,C 180,E1 20976.68,E2 20976.68} C_VEL
LIN {X 0,Y 575.904,Z 1172.237,A -85,B 0,C 180,E1 20974.581,E2 20974.581} C_VEL
LIN {X 0,Y 575.91,Z 1174.108,A -85,B 0,C 180,E1 20972.488,E2 20972.488} C_VEL
LIN {X 0,Y 575.915,Z 1174.993,A -85,B 0,C 180,E1 20970,E2 20970} C_VEL
LIN {X 0,Y 575.914,Z 1174.173,A -85,B 0,C 180,E1 20967.513,E2 20967.513} C_VEL
LIN {X 0,Y 575.903,Z 1172.341,A -85,B 0,C 180,E1 20965.419,E2 20965.419} C_VEL
LIN {X 0,Y 575.946,Z 1169.42,A -85,B 0,C 180,E1 20963.321,E2 20963.321} C_VEL
LIN {X 0,Y 576.066,Z 1164.542,A -85,B 0,C 180,E1 20960.812,E2 20960.812} C_VEL
LIN {X 0,Y 576.279,Z 1158.119,A -85,B 0,C 180,E1 20958.389,E2 20958.389} C_VEL
LIN {X 0,Y 576.606,Z 1151.606,A -85,B 0,C 180,E1 20956.359,E2 20956.359} C_VEL
LIN {X 0,Y 577.114,Z 1143.529,A -85,B 0,C 180,E1 20954.216,E2 20954.216} C_VEL
LIN {X 0,Y 578.058,Z 1131.564,A -85,B 0,C 180,E1 20951.547,E2 20951.547} C_VEL
LIN {X 0,Y 579.07,Z 1120.761,A -85,B 0,C 180,E1 20949.481,E2 20949.481} C_VEL
LIN {X 0,Y 580.475,Z 1107.868,A -85,B 0,C 180,E1 20947.304,E2 20947.304} C_VEL
LIN {X 0,Y 582.294,Z 1092.219,A -85,B 0,C 180,E1 20945.013,E2 20945.013} C_VEL
LIN {X 0,Y 584.047,Z 1078.55,A -85,B 0,C 180,E1 20943.24,E2 20943.24} C_VEL
LIN {X 0,Y 586.494,Z 1060.593,A -85,B 0,C 180,E1 20941.153,E2 20941.153} C_VEL
LIN {X 0,Y 589.224,Z 1041.952,A -85,B 0,C 180,E1 20939.228,E2 20939.228} C_VEL
LIN {X 0,Y 591.707,Z 1025.649,A -85,B 0,C 180,E1 20937.725,E2 20937.725} C_VEL
LIN {X 0,Y 594.903,Z 1004.919,A -85,B 0,C 180,E1 20936.024,E2 20936.024} C_VEL
LIN {X 0,Y 597.979,Z 983.614,A -85,B 0,C 180,E1 20934.521,E2 20934.521} C_VEL
LIN {X 0,Y 600.745,Z 963.991,A -85,B 0,C 180,E1 20933.308,E2 20933.308} C_VEL
LIN {X 0,Y 604.019,Z 939.244,A -85,B 0,C 180,E1 20931.996,E2 20931.996} C_VEL
LIN {X 0,Y 606.426,Z 918.729,A -85,B 0,C 180,E1 20931.083,E2 20931.083} C_VEL
LIN {X 0,Y 608.574,Z 898.137,A -85,B 0,C 180,E1 20930.305,E2 20930.305} C_VEL
LIN {X 0,Y 610.87,Z 873.184,A -85,B 0,C 180,E1 20929.535,E2 20929.535} C_VEL
LIN {X 0,Y 612.476,Z 849.248,A -85,B 0,C 180,E1 20928.977,E2 20928.977} C_VEL
LIN {X 0,Y 613.525,Z 827.736,A -85,B 0,C 180,E1 20928.6,E2 20928.6} C_VEL
LIN {X 0,Y 618.839,Z 609.565,A -85,B 0,C 180,E1 20925.657,E2 20925.657} C_VEL
LIN {X 0,Y 623.099,Z 439.733,A -85,B 0,C 180,E1 20923.322,E2 20923.322} C_VEL
LIN {X 0,Y 616.095,Z 405.478,A -85,B 0,C 180,E1 20921.979,E2 20921.979} C_VEL
LIN {X 0,Y 606.171,Z 390.373,A -85,B 0,C 180,E1 20920.535,E2 20920.535} C_VEL
LIN {X 0,Y 598.371,Z 373.398,A -85,B 0,C 180,E1 20918.008,E2 20918.008} C_VEL
LIN {X 0,Y 591.7,Z 360.021,A -85,B 0,C 180,E1 20915.781,E2 20915.781} C_VEL
LIN {X 0,Y 586.537,Z 350.256,A -85,B 0,C 180,E1 20913.997,E2 20913.997} C_VEL
LIN {X 0,Y 584.367,Z 346.025,A -85,B 0,C 180,E1 20913.199,E2 20913.199} C_VEL
LIN {X 0,Y 581.863,Z 341.425,A -85,B 0,C 180,E1 20912.28,E2 20912.28} C_VEL
LIN {X 0,Y 579.371,Z 336.754,A -85,B 0,C 180,E1 20911.321,E2 20911.321} C_VEL
LIN {X 0,Y 577.51,Z 333.472,A -85,B 0,C 180,E1 20910.599,E2 20910.599} C_VEL
LIN {X 0,Y 577.31,Z 332.503,A -85,B 0,C 180,E1 20910.381,E2 20910.381} C_VEL
LIN {X 0,Y 577.317,Z 332.288,A -85,B 0,C 180,E1 20907.317,E2 20907.317} C_VEL
LIN {X 0,Y 577.301,Z 332.265,A -85,B 0,C 180,E1 20904.018,E2 20904.018} C_VEL
LIN {X 0,Y 577.295,Z 332.316,A -85,B 0,C 180,E1 20900.691,E2 20900.691} C_VEL
LIN {X 0,Y 577.309,Z 332.271,A -85,B 0,C 180,E1 20897.436,E2 20897.436} C_VEL
LIN {X 0,Y 577.294,Z 332.29,A -85,B 0,C 180,E1 20894.238,E2 20894.238} C_VEL
LIN {X 0,Y 577.308,Z 332.282,A -85,B 0,C 180,E1 20890.983,E2 20890.983} C_VEL
LIN {X 0,Y 577.314,Z 332.27,A -85,B 0,C 180,E1 20887.664,E2 20887.664} C_VEL
LIN {X 0,Y 577.307,Z 332.305,A -85,B 0,C 180,E1 20884.271,E2 20884.271} C_VEL
LIN {X 0,Y 577.292,Z 332.267,A -85,B 0,C 180,E1 20881.092,E2 20881.092} C_VEL
LIN {X 0,Y 577.313,Z 332.308,A -85,B 0,C 180,E1 20877.816,E2 20877.816} C_VEL
LIN {X 0,Y 577.299,Z 332.263,A -85,B 0,C 180,E1 20874.534,E2 20874.534} C_VEL
LIN {X 0,Y 577.295,Z 332.317,A -85,B 0,C 180,E1 20871.233,E2 20871.233} C_VEL
LIN {X 0,Y 577.313,Z 332.258,A -85,B 0,C 180,E1 20868.004,E2 20868.004} C_VEL
LIN {X 0,Y 577.279,Z 332.322,A -85,B 0,C 180,E1 20864.838,E2 20864.838} C_VEL
LIN {X 0,Y 577.315,Z 332.262,A -85,B 0,C 180,E1 20861.626,E2 20861.626} C_VEL
LIN {X 0,Y 577.271,Z 332.302,A -85,B 0,C 180,E1 20858.454,E2 20858.454} C_VEL
LIN {X 0,Y 577.293,Z 332.291,A -85,B 0,C 180,E1 20855.172,E2 20855.172} C_VEL
LIN {X 0,Y 577.269,Z 332.271,A -85,B 0,C 180,E1 20852.117,E2 20852.117} C_VEL
LIN {X 0,Y 577.331,Z 332.544,A -85,B 0,C 180,E1 20851.162,E2 20851.162} C_VEL
LIN {X 0,Y 578.61,Z 335.848,A -85,B 0,C 180,E1 20850.494,E2 20850.494} C_VEL
LIN {X 0,Y 580.134,Z 337.837,A -85,B 0,C 180,E1 20850.011,E2 20850.011} C_VEL
LIN {X 0,Y 582.243,Z 341.844,A -85,B 0,C 180,E1 20849.219,E2 20849.219} C_VEL
LIN {X 0,Y 585.027,Z 346.862,A -85,B 0,C 180,E1 20848.236,E2 20848.236} C_VEL
LIN {X 0,Y 590.496,Z 356.792,A -85,B 0,C 180,E1 20846.436,E2 20846.436} C_VEL
LIN {X 0,Y 603.617,Z 374.173,A -85,B 0,C 180,E1 20844.39,E2 20844.39} C_VEL
LIN {X 0,Y 616.311,Z 391.715,A -85,B 0,C 180,E1 20842.57,E2 20842.57} C_VEL
LIN {X 0,Y 628.123,Z 409.047,A -85,B 0,C 180,E1 20840.984,E2 20840.984} C_VEL
LIN {X 0,Y 622.711,Z 608.932,A -85,B 0,C 180,E1 20838.145,E2 20838.145} C_VEL
LIN {X 0,Y 617.395,Z 826.022,A -85,B 0,C 180,E1 20835.153,E2 20835.153} C_VEL
LIN {X 0,Y 616.216,Z 849.672,A -85,B 0,C 180,E1 20834.737,E2 20834.737} C_VEL
LIN {X 0,Y 614.227,Z 878.839,A -85,B 0,C 180,E1 20834.039,E2 20834.039} C_VEL
LIN {X 0,Y 612.38,Z 900.903,A -85,B 0,C 180,E1 20833.366,E2 20833.366} C_VEL
LIN {X 0,Y 610.384,Z 921.924,A -85,B 0,C 180,E1 20832.605,E2 20832.605} C_VEL
LIN {X 0,Y 608.185,Z 942.928,A -85,B 0,C 180,E1 20831.72,E2 20831.72} C_VEL
LIN {X 0,Y 606.182,Z 959.674,A -85,B 0,C 180,E1 20830.907,E2 20830.907} C_VEL
LIN {X 0,Y 603.546,Z 979.421,A -85,B 0,C 180,E1 20829.814,E2 20829.814} C_VEL
LIN {X 0,Y 600.184,Z 1003.431,A -85,B 0,C 180,E1 20828.296,E2 20828.296} C_VEL
LIN {X 0,Y 596.944,Z 1024.884,A -85,B 0,C 180,E1 20826.725,E2 20826.725} C_VEL
LIN {X 0,Y 594.204,Z 1042.825,A -85,B 0,C 180,E1 20825.252,E2 20825.252} C_VEL
LIN {X 0,Y 591.552,Z 1060.156,A -85,B 0,C 180,E1 20823.669,E2 20823.669} C_VEL
LIN {X 0,Y 588.525,Z 1080.339,A -85,B 0,C 180,E1 20821.609,E2 20821.609} C_VEL
LIN {X 0,Y 585.85,Z 1098.46,A -85,B 0,C 180,E1 20819.49,E2 20819.49} C_VEL
LIN {X 0,Y 583.723,Z 1113.38,A -85,B 0,C 180,E1 20817.548,E2 20817.548} C_VEL
LIN {X 0,Y 581.679,Z 1129.283,A -85,B 0,C 180,E1 20815.233,E2 20815.233} C_VEL
LIN {X 0,Y 579.853,Z 1144.403,A -85,B 0,C 180,E1 20812.698,E2 20812.698} C_VEL
LIN {X 0,Y 578.642,Z 1155.781,A -85,B 0,C 180,E1 20810.535,E2 20810.535} C_VEL
LIN {X 0,Y 577.699,Z 1166.363,A -85,B 0,C 180,E1 20808.256,E2 20808.256} C_VEL
LIN {X 0,Y 576.865,Z 1177.389,A -85,B 0,C 180,E1 20805.479,E2 20805.479} C_VEL
LIN {X 0,Y 576.432,Z 1185.173,A -85,B 0,C 180,E1 20803.134,E2 20803.134} C_VEL
LIN {X 0,Y 576.142,Z 1191.612,A -85,B 0,C 180,E1 20800.798,E2 20800.798} C_VEL
LIN {X 0,Y 575.999,Z 1197.151,A -85,B 0,C 180,E1 20798.284,E2 20798.284} C_VEL
LIN {X 0,Y 575.933,Z 1201.427,A -85,B 0,C 180,E1 20795.579,E2 20795.579} C_VEL
LIN {X 0,Y 575.917,Z 1203.851,A -85,B 0,C 180,E1 20793.085,E2 20793.085} C_VEL
LIN {X 0,Y 575.905,Z 1204.804,A -85,B 0,C 180,E1 20790.895,E2 20790.895} C_VEL
LIN {X 0,Y 575.915,Z 1204.736,A -85,B 0,C 180,E1 20788.806,E2 20788.806} C_VEL
LIN {X 0,Y 575.913,Z 1203.509,A -85,B 0,C 180,E1 20786.416,E2 20786.416} C_VEL
LIN {X 0,Y 575.947,Z 1200.336,A -85,B 0,C 180,E1 20783.621,E2 20783.621} C_VEL
LIN {X 0,Y 576.025,Z 1195.922,A -85,B 0,C 180,E1 20781.113,E2 20781.113} C_VEL
LIN {X 0,Y 576.176,Z 1190.582,A -85,B 0,C 180,E1 20778.792,E2 20778.792} C_VEL
LIN {X 0,Y 576.568,Z 1182.683,A -85,B 0,C 180,E1 20776.051,E2 20776.051} C_VEL
LIN {X 0,Y 577.161,Z 1173.11,A -85,B 0,C 180,E1 20773.39,E2 20773.39} C_VEL
LIN {X 0,Y 577.892,Z 1164.07,A -85,B 0,C 180,E1 20771.227,E2 20771.227} C_VEL
LIN {X 0,Y 578.926,Z 1153.205,A -85,B 0,C 180,E1 20768.946,E2 20768.946} C_VEL
LIN {X 0,Y 580.563,Z 1138.271,A -85,B 0,C 180,E1 20766.233,E2 20766.233} C_VEL
LIN {X 0,Y 582.163,Z 1125.078,A -85,B 0,C 180,E1 20764.135,E2 20764.135} C_VEL
LIN {X 0,Y 584.064,Z 1111.065,A -85,B 0,C 180,E1 20762.137,E2 20762.137} C_VEL
LIN {X 0,Y 586.668,Z 1092.847,A -85,B 0,C 180,E1 20759.816,E2 20759.816} C_VEL
LIN {X 0,Y 589.383,Z 1074.493,A -85,B 0,C 180,E1 20757.776,E2 20757.776} C_VEL
LIN {X 0,Y 591.898,Z 1057.931,A -85,B 0,C 180,E1 20756.119,E2 20756.119} C_VEL
LIN {X 0,Y 594.594,Z 1040.382,A -85,B 0,C 180,E1 20754.538,E2 20754.538} C_VEL
LIN {X 0,Y 598.03,Z 1017.906,A -85,B 0,C 180,E1 20752.737,E2 20752.737} C_VEL
LIN {X 0,Y 601.155,Z 996.218,A -85,B 0,C 180,E1 20751.228,E2 20751.228} C_VEL
LIN {X 0,Y 603.896,Z 976.713,A -85,B 0,C 180,E1 20750.028,E2 20750.028} C_VEL
LIN {X 0,Y 606.435,Z 957.661,A -85,B 0,C 180,E1 20748.988,E2 20748.988} C_VEL
LIN {X 0,Y 608.24,Z 942.44,A -85,B 0,C 180,E1 20748.258,E2 20748.258} C_VEL
LIN {X 0,Y 610.452,Z 921.243,A -85,B 0,C 180,E1 20747.368,E2 20747.368} C_VEL
LIN {X 0,Y 612.513,Z 899.505,A -85,B 0,C 180,E1 20746.587,E2 20746.587} C_VEL
LIN {X 0,Y 614.739,Z 872.634,A -85,B 0,C 180,E1 20745.792,E2 20745.792} C_VEL
LIN {X 0,Y 616.347,Z 847.096,A -85,B 0,C 180,E1 20745.213,E2 20745.213} C_VEL
LIN {X 0,Y 617.437,Z 824.871,A -85,B 0,C 180,E1 20744.83,E2 20744.83} C_VEL
LIN {X 0,Y 622.813,Z 603.588,A -85,B 0,C 180,E1 20741.784,E2 20741.784} C_VEL
LIN {X 0,Y 628.102,Z 408.839,A -85,B 0,C 180,E1 20739.011,E2 20739.011} C_VEL
LIN {X 0,Y 613.858,Z 388.328,A -85,B 0,C 180,E1 20737.092,E2 20737.092} C_VEL
LIN {X 0,Y 601.339,Z 371.083,A -85,B 0,C 180,E1 20735.273,E2 20735.273} C_VEL
LIN {X 0,Y 590.223,Z 356.468,A -85,B 0,C 180,E1 20733.523,E2 20733.523} C_VEL
LIN {X 0,Y 584.995,Z 346.824,A -85,B 0,C 180,E1 20731.766,E2 20731.766} C_VEL
LIN {X 0,Y 582.803,Z 342.705,A -85,B 0,C 180,E1 20730.977,E2 20730.977} C_VEL
LIN {X 0,Y 580.319,Z 338.36,A -85,B 0,C 180,E1 20730.092,E2 20730.092} C_VEL
LIN {X 0,Y 578.868,Z 336.206,A -85,B 0,C 180,E1 20729.605,E2 20729.605} C_VEL
LIN {X 0,Y 577.335,Z 332.593,A -85,B 0,C 180,E1 20728.867,E2 20728.867} C_VEL
LIN {X 0,Y 577.257,Z 332.28,A -85,B 0,C 180,E1 20727.305,E2 20727.305} C_VEL
LIN {X 0,Y 577.301,Z 332.271,A -85,B 0,C 180,E1 20724.111,E2 20724.111} C_VEL
LIN {X 0,Y 577.278,Z 332.32,A -85,B 0,C 180,E1 20721,E2 20721} C_VEL
LIN {X 0,Y 577.279,Z 332.265,A -85,B 0,C 180,E1 20717.645,E2 20717.645} C_VEL
LIN {X 0,Y 577.324,Z 332.308,A -85,B 0,C 180,E1 20714.442,E2 20714.442} C_VEL
LIN {X 0,Y 577.275,Z 332.273,A -85,B 0,C 180,E1 20711.186,E2 20711.186} C_VEL
LIN {X 0,Y 577.318,Z 332.294,A -85,B 0,C 180,E1 20707.964,E2 20707.964} C_VEL
LIN {X 0,Y 577.293,Z 332.281,A -85,B 0,C 180,E1 20704.669,E2 20704.669} C_VEL
LIN {X 0,Y 577.299,Z 332.281,A -85,B 0,C 180,E1 20701.29,E2 20701.29} C_VEL
LIN {X 0,Y 577.309,Z 332.289,A -85,B 0,C 180,E1 20698.015,E2 20698.015} C_VEL
LIN {X 0,Y 577.293,Z 332.274,A -85,B 0,C 180,E1 20694.815,E2 20694.815} C_VEL
LIN {X 0,Y 577.304,Z 332.29,A -85,B 0,C 180,E1 20691.634,E2 20691.634} C_VEL
LIN {X 0,Y 577.305,Z 332.266,A -85,B 0,C 180,E1 20688.41,E2 20688.41} C_VEL
LIN {X 0,Y 577.322,Z 332.312,A -85,B 0,C 180,E1 20685.045,E2 20685.045} C_VEL
LIN {X 0,Y 577.294,Z 332.263,A -85,B 0,C 180,E1 20681.73,E2 20681.73} C_VEL
LIN {X 0,Y 577.314,Z 332.316,A -85,B 0,C 180,E1 20678.444,E2 20678.444} C_VEL
LIN {X 0,Y 577.289,Z 332.275,A -85,B 0,C 180,E1 20675.173,E2 20675.173} C_VEL
LIN {X 0,Y 577.306,Z 332.272,A -85,B 0,C 180,E1 20671.894,E2 20671.894} C_VEL
LIN {X 0,Y 577.322,Z 332.566,A -85,B 0,C 180,E1 20669.482,E2 20669.482} C_VEL
LIN {X 0,Y 578.707,Z 335.941,A -85,B 0,C 180,E1 20668.779,E2 20668.779} C_VEL
LIN {X 0,Y 580.157,Z 338.036,A -85,B 0,C 180,E1 20668.287,E2 20668.287} C_VEL
LIN {X 0,Y 581.961,Z 341.544,A -85,B 0,C 180,E1 20667.584,E2 20667.584} C_VEL
LIN {X 0,Y 585.569,Z 348.285,A -85,B 0,C 180,E1 20666.26,E2 20666.26} C_VEL
LIN {X 0,Y 590.563,Z 357.896,A -85,B 0,C 180,E1 20664.497,E2 20664.497} C_VEL
LIN {X 0,Y 596.445,Z 369.563,A -85,B 0,C 180,E1 20662.516,E2 20662.516} C_VEL
LIN {X 0,Y 604.084,Z 385.614,A -85,B 0,C 180,E1 20660.042,E2 20660.042} C_VEL
LIN {X 0,Y 606.9,Z 391.672,A -85,B 0,C 180,E1 20659.228,E2 20659.228} C_VEL
LIN {X 0,Y 616.301,Z 405.858,A -85,B 0,C 180,E1 20657.897,E2 20657.897} C_VEL
LIN {X 0,Y 623.147,Z 440.479,A -85,B 0,C 180,E1 20656.568,E2 20656.568} C_VEL
LIN {X 0,Y 618.786,Z 611.389,A -85,B 0,C 180,E1 20654.228,E2 20654.228} C_VEL
LIN {X 0,Y 617.908,Z 619.096,A -85,B 0,C 180,E1 20654.191,E2 20654.191} C_VEL
LIN {X 0,Y 613.076,Z 639.732,A -85,B 0,C 180,E1 20654.337,E2 20654.337} C_VEL
LIN {X 0,Y 612.398,Z 646.343,A -85,B 0,C 180,E1 20654.298,E2 20654.298} C_VEL
LIN {X 0,Y 607.696,Z 830.551,A -85,B 0,C 180,E1 20651.796,E2 20651.796} C_VEL
LIN {X 0,Y 606.284,Z 856.471,A -85,B 0,C 180,E1 20651.319,E2 20651.319} C_VEL
LIN {X 0,Y 604.32,Z 881.261,A -85,B 0,C 180,E1 20650.677,E2 20650.677} C_VEL
LIN {X 0,Y 602.345,Z 902.102,A -85,B 0,C 180,E1 20650.003,E2 20650.003} C_VEL
LIN {X 0,Y 599.64,Z 926.737,A -85,B 0,C 180,E1 20649.031,E2 20649.031} C_VEL
LIN {X 0,Y 596.696,Z 949.119,A -85,B 0,C 180,E1 20647.951,E2 20647.951} C_VEL
LIN {X 0,Y 593.992,Z 968.208,A -85,B 0,C 180,E1 20646.883,E2 20646.883} C_VEL
LIN {X 0,Y 590.764,Z 989.945,A -85,B 0,C 180,E1 20645.488,E2 20645.488} C_VEL
LIN {X 0,Y 587.326,Z 1011.321,A -85,B 0,C 180,E1 20643.886,E2 20643.886} C_VEL
LIN {X 0,Y 584.549,Z 1028.499,A -85,B 0,C 180,E1 20642.429,E2 20642.429} C_VEL
LIN {X 0,Y 581.392,Z 1048.216,A -85,B 0,C 180,E1 20640.545,E2 20640.545} C_VEL
LIN {X 0,Y 578.571,Z 1065.878,A -85,B 0,C 180,E1 20638.601,E2 20638.601} C_VEL
LIN {X 0,Y 576.149,Z 1082.139,A -85,B 0,C 180,E1 20636.599,E2 20636.599} C_VEL
LIN {X 0,Y 573.905,Z 1098.995,A -85,B 0,C 180,E1 20634.278,E2 20634.278} C_VEL
LIN {X 0,Y 572.316,Z 1111.78,A -85,B 0,C 180,E1 20632.279,E2 20632.279} C_VEL
LIN {X 0,Y 570.96,Z 1124.286,A -85,B 0,C 180,E1 20630.075,E2 20630.075} C_VEL
LIN {X 0,Y 569.789,Z 1136.486,A -85,B 0,C 180,E1 20627.568,E2 20627.568} C_VEL
LIN {X 0,Y 569.094,Z 1145.2,A -85,B 0,C 180,E1 20625.49,E2 20625.49} C_VEL
LIN {X 0,Y 568.568,Z 1153.413,A -85,B 0,C 180,E1 20623.216,E2 20623.216} C_VEL
LIN {X 0,Y 568.183,Z 1161.265,A -85,B 0,C 180,E1 20620.546,E2 20620.546} C_VEL
LIN {X 0,Y 568.028,Z 1166.248,A -85,B 0,C 180,E1 20618.395,E2 20618.395} C_VEL
LIN {X 0,Y 567.95,Z 1170.076,A -85,B 0,C 180,E1 20616.267,E2 20616.267} C_VEL
LIN {X 0,Y 567.912,Z 1173.145,A -85,B 0,C 180,E1 20613.836,E2 20613.836} C_VEL
LIN {X 0,Y 567.91,Z 1174.722,A -85,B 0,C 180,E1 20611.211,E2 20611.211} C_VEL
LIN {X 0,Y 567.904,Z 1174.812,A -85,B 0,C 180,E1 20609.092,E2 20609.092} C_VEL
LIN {X 0,Y 567.906,Z 1173.9,A -85,B 0,C 180,E1 20607.074,E2 20607.074} C_VEL
LIN {X 0,Y 567.924,Z 1171.659,A -85,B 0,C 180,E1 20604.747,E2 20604.747} C_VEL
LIN {X 0,Y 567.997,Z 1167.452,A -85,B 0,C 180,E1 20602.108,E2 20602.108} C_VEL
LIN {X 0,Y 568.112,Z 1162.761,A -85,B 0,C 180,E1 20599.966,E2 20599.966} C_VEL
LIN {X 0,Y 568.379,Z 1156.903,A -85,B 0,C 180,E1 20597.813,E2 20597.813} C_VEL
LIN {X 0,Y 568.85,Z 1148.768,A -85,B 0,C 180,E1 20595.339,E2 20595.339} C_VEL
LIN {X 0,Y 569.585,Z 1138.717,A -85,B 0,C 180,E1 20592.848,E2 20592.848} C_VEL
LIN {X 0,Y 570.473,Z 1128.983,A -85,B 0,C 180,E1 20590.761,E2 20590.761} C_VEL
LIN {X 0,Y 571.857,Z 1116.128,A -85,B 0,C 180,E1 20588.351,E2 20588.351} C_VEL
LIN {X 0,Y 573.458,Z 1102.379,A -85,B 0,C 180,E1 20586.14,E2 20586.14} C_VEL
